TYPE "UDT_ModuleState"
TITLE = UDT_ModuleState
VERSION : 0.1
//User-defined structure of module states.
   STRUCT
      Configured { ExternalAccessible := 'False'; ExternalVisible := 'False'; ExternalWritable := 'False'} : Bool;   // Module configured
      Exist { ExternalAccessible := 'False'; ExternalVisible := 'False'; ExternalWritable := 'False'} : Bool;   // Module exist
      Error { ExternalAccessible := 'False'; ExternalVisible := 'False'; ExternalWritable := 'False'} : Bool;   // Module has error
   END_STRUCT;

END_TYPE

TYPE "UDT_DeviceState"
TITLE = UDT_DeviceState
VERSION : 0.1
//User-defined structure of device states.
   STRUCT
      Configure { ExternalAccessible := 'False'; ExternalVisible := 'False'; ExternalWritable := 'False'} : Bool;   // Device configured in TIA Portal hardware
      Exist { ExternalAccessible := 'False'; ExternalVisible := 'False'; ExternalWritable := 'False'} : Bool;   // Device physically connected
      Error { ExternalAccessible := 'False'; ExternalVisible := 'False'; ExternalWritable := 'False'} : Bool;   // Device has an error
      ProfinetNumber : UInt;   // Profinet slave number
      HW_ID : UInt;   // Device's HW_ID
      PNDeviceName : String;   // Device's project name
   END_STRUCT;

END_TYPE

TYPE "UDT_ProfinetDevice"
TITLE = UDT_ProfinetDevice
VERSION : 0.1
//User-defined structure of profinet device state.
   STRUCT
      DeviceState : "UDT_DeviceState";   // Device state
      Module { S7_SetPoint := 'False'} : Array[0..31] of "UDT_ModuleState";   // Modules
   END_STRUCT;

END_TYPE

TYPE "UDT_GINWCS"
VERSION : 0.1
   STRUCT
      ActionTaken : String;   // Location code value that describes the actual disposition of the package
      Destination1 : String[20];   // Location code value that describes where the package should go (Diverter Number)
      Destination2 : String[20];   // Location code value that describes where the package should go (Diverter Number)
      Destination3 : String[20];   // Location code value that describes where the package should go (Diverter Number)
      Destination4 : String[20];   // Location code value that describes where the package should go (Diverter Number)
      Destination5 : String[20];   // Location code value that describes where the package should go (Diverter Number)
      ReasonCode : String[2];   // Management Code value that describes the result of attempting to route the package to the Destination
      Barcode1 : String;   // Barcode identifier code
      Barcode2 : String;
      Barcode3 : String;
      Barcode4 : String;
   END_STRUCT;

END_TYPE

TYPE "UDT_ProfinetNetwork"
TITLE = UDT_ProfinetNetwork
VERSION : 0.1
//User-defined structure of profinet network state.
   STRUCT
      DeviceStatus : Array[0..512] of "UDT_ProfinetDevice";   // Profinet device status
   END_STRUCT;

END_TYPE

TYPE "UDT_GINWES"
VERSION : 0.1
   STRUCT
      Barcode : String[40];
   END_STRUCT;

END_TYPE

TYPE "UDT_GINDHL"
VERSION : 0.1
   STRUCT
      ObjectID : String[10];   // Object ID
      VID : String[16];   // Virtual Item Identifier (VID)
      PieceID : String[40];   // Piece ID barcodes
      SortStrategy : String[1];   // Sort Strategy 1 - Highest priority available , 2 - Nearest
      ParcelReject { ExternalAccessible := 'False'; ExternalVisible := 'False'; ExternalWritable := 'False'} : Bool;   // True - Parcel reject
      Destination : Array[1..6] of Struct   // Destination
         ID : UInt;   // ID
         SortCommandActive { ExternalAccessible := 'False'; ExternalVisible := 'False'; ExternalWritable := 'False'} : Bool;   // Sort command
         ParcelSorted { ExternalAccessible := 'False'; ExternalVisible := 'False'; ExternalWritable := 'False'} : Bool;   // Parcel sorted
         Rejected { ExternalAccessible := 'False'; ExternalVisible := 'False'; ExternalWritable := 'False'} : Bool;   // Parcel rejected
         Reason : Int;   // Reason
      END_STRUCT;
      ParcelLocation : Struct   // Parcel Location
         Current : UInt;   // Current
         Last : UInt;   // Last
         Sort : UInt;   // Sort
      END_STRUCT;
      MFCMessage : Struct   // MFC Sort messages
         Sent : Struct   // Messages sent from the PLC to the MFC system
            SortResult { ExternalAccessible := 'False'; ExternalVisible := 'False'; ExternalWritable := 'False'} : Bool;   // Message Sort Result
            VIDResponse { ExternalAccessible := 'False'; ExternalVisible := 'False'; ExternalWritable := 'False'} : Bool;   // Message VID Response
            ScanReset { ExternalAccessible := 'False'; ExternalVisible := 'False'; ExternalWritable := 'False'} : Bool;   // Message Scan Reset
            XrayResult { ExternalAccessible := 'False'; ExternalVisible := 'False'; ExternalWritable := 'False'} : Bool;   // Message Xray result
            ParcelRegInfo { ExternalAccessible := 'False'; ExternalVisible := 'False'; ExternalWritable := 'False'} : Bool;   // Message Xray registration info
         END_STRUCT;
         Received : Struct   // Messages received from the MFC system to the PLC
            RejectParcel { ExternalAccessible := 'False'; ExternalVisible := 'False'; ExternalWritable := 'False'} : Bool;   // Message Reject Parcel
            Destination { ExternalAccessible := 'False'; ExternalVisible := 'False'; ExternalWritable := 'False'} : Bool;   // Message Destination
            DestinationResent { ExternalAccessible := 'False'; ExternalVisible := 'False'; ExternalWritable := 'False'} : Bool;   // Message Destination Resent
            TemporaryParcelIdentifier { ExternalAccessible := 'False'; ExternalVisible := 'False'; ExternalWritable := 'False'} : Bool;   // Message Temporary Parcel Identifier
            XrayRegistrationInfo { ExternalAccessible := 'False'; ExternalVisible := 'False'; ExternalWritable := 'False'} : Bool;
         END_STRUCT;
      END_STRUCT;
      Xray : Struct   // Xray data structure
         RoutingCode : String[2];   // Routing code
         Group : String[1];   // The group field is used to identify the group of the operator decisions came from in a
         Level : String[1];   // Level field is used to identify which level the operator decision came from in a
         Result : String[1];   // Results can be indicated with the following:A = Accept, R = Reject, U = Unavailable (Timeout), Z = High Threat
         BagIDMessage : Struct   // Message from PLC to Xray
            MessagePrepared { ExternalAccessible := 'False'; ExternalVisible := 'False'; ExternalWritable := 'False'} : Bool;   // The message is prepared and ready to send
            WrongMessageStructure { ExternalAccessible := 'False'; ExternalVisible := 'False'; ExternalWritable := 'False'} : Bool;   // The message has wrong structure
            Sent { ExternalAccessible := 'False'; ExternalVisible := 'False'; ExternalWritable := 'False'} : Bool;   // The message sent by PLC to Xray
            SentTime : String;   // Time when message sent by PLC to Xray
            NotSent { ExternalAccessible := 'False'; ExternalVisible := 'False'; ExternalWritable := 'False'} : Bool;   // The message was not sent from the PLC
            Received { ExternalAccessible := 'False'; ExternalVisible := 'False'; ExternalWritable := 'False'} : Bool;   // The message received by Xray
            TimeReceived : String;   // Time when message received by Xray
            NotReceived { ExternalAccessible := 'False'; ExternalVisible := 'False'; ExternalWritable := 'False'} : Bool;   // The message did not reach Xray
         END_STRUCT;
         DecisionMessage : Struct   // Message from Xray to PLC
            Received { ExternalAccessible := 'False'; ExternalVisible := 'False'; ExternalWritable := 'False'} : Bool;   // The message received by PLC
            ReceivedTime : String;   // The message received by PLC
            NotReceivedOnTime { ExternalAccessible := 'False'; ExternalVisible := 'False'; ExternalWritable := 'False'} : Bool;   // The message did not reach PLC
         END_STRUCT;
      END_STRUCT;
   END_STRUCT;

END_TYPE

TYPE "UDT_GINUPS"
VERSION : 0.1
   STRUCT
      TRKNUM : String[18];   // Tracking number
      PKGUID : String[32];   // Package ID
      MSGID : String[32];   // Message ID
      Length : Int;   // Camera Length in mm
      Width : Int;   // Camera Width in mm
      Height : Int;   // Camera Height in mm
      Weight : DInt;   // Weight in g
      IDCreated { ExternalAccessible := 'False'; ExternalVisible := 'False'; ExternalWritable := 'False'} : Bool;   // Byte 1, Bit 0 - PLCID created or TrayID Read
      DimDataRcv { ExternalAccessible := 'False'; ExternalVisible := 'False'; ExternalWritable := 'False'} : Bool;   // Byte 1, Bit 1 - Package Dimensional Data Received via Camera Scan Data Message
      PkgWrongInduct { ExternalAccessible := 'False'; ExternalVisible := 'False'; ExternalWritable := 'False'} : Bool;   // Byte 1, Bit 2 - Package Did NOT Induct Properly (Non-Tray Systems)
      IDCalcFromCamID { ExternalAccessible := 'False'; ExternalVisible := 'False'; ExternalWritable := 'False'} : Bool;   // Byte 2, Bit 0 - PLCID/TrayID Calculated From CamID
      UnknownParcelID { ExternalAccessible := 'False'; ExternalVisible := 'False'; ExternalWritable := 'False'} : Bool;   // Byte 2, Bit 4 - Unknown Parcel ID
      UndefinedProblem { ExternalAccessible := 'False'; ExternalVisible := 'False'; ExternalWritable := 'False'} : Bool;   // Byte 2, Bit 5 - Un-Defined Problem
      UnrecognizedCmd { ExternalAccessible := 'False'; ExternalVisible := 'False'; ExternalWritable := 'False'} : Bool;   // Byte 2, Bit 6 - Un-recognized command
      SorterInMainteneceMode { ExternalAccessible := 'False'; ExternalVisible := 'False'; ExternalWritable := 'False'} : Bool;   // Byte 2, Bit 7 - Sorter in Maintenance/Commissioning Mode
      DestUserSusp { ExternalAccessible := 'False'; ExternalVisible := 'False'; ExternalWritable := 'False'} : Bool;   // Byte 3, Bit 3 - Destination User Suspended
      SorterNotSynch { ExternalAccessible := 'False'; ExternalVisible := 'False'; ExternalWritable := 'False'} : Bool;   // Byte 3, Bit 6 - Sorter NOT Synchronized (Tilt Tray Systems)
      PkgDetAtVerCheckPoint { ExternalAccessible := 'False'; ExternalVisible := 'False'; ExternalWritable := 'False'} : Bool;   // Byte 4, Bit 0 - Package Detected at Verification Check Point
      ChuteFullAftrAlterDest { ExternalAccessible := 'False'; ExternalVisible := 'False'; ExternalWritable := 'False'} : Bool;   // Byte 4, Bit 7 - Preferred chute full after passed alternate destination
      ChuteNotAvailAfterAlterDest { ExternalAccessible := 'False'; ExternalVisible := 'False'; ExternalWritable := 'False'} : Bool;   // Byte 5, Bit 0 - Preferred chute not available after passed alternate destination
      PLCRedirected { ExternalAccessible := 'False'; ExternalVisible := 'False'; ExternalWritable := 'False'} : Bool;   // Byte 5, Bit 2 - PLC Redirected
      ThreatParcel { ExternalAccessible := 'False'; ExternalVisible := 'False'; ExternalWritable := 'False'} : Bool;   // Threat parcel
   END_STRUCT;

END_TYPE

TYPE "UDT_GINFedEx"
VERSION : 0.1
   STRUCT
      Timestamp : String[17];   // Local time timestamp
      TimeZoneDesignator : String[5];   // Time zone designator
      PackageEntrancePoint : String[14];   // Entrance point, where LLC starts tracking the parcel.
      PackageEntranceState : String[1];   // Entrance state
      PackageExitPoint : String[14];   // Exit point name, where LLC reports the last known tracking point.
      PackageExitState : String[1];   // Exit point state when LLC reports the last known tracking point.
      PalletType : String[2];   // Pallet code for different type of pallets on the market
      Mask : String[1];   // Flag to indicate that a pallet has been mask.
      CellNumber : String[4];   // Tray/Cell number (for loop sorters) or generated by LLC (on line sorters).
      CellsOccupied : String[1];   // Cells occupied by the piece for loop sorters.
      ImageID : String[6];   // Image ID number created by the ADC system.
      ScanUnitType : String[1];   // Scan unit type
      ADCSystemID : String[15];   // Number assigned by the ADC system
      PackageID : String[15];   // Number assigned by the LLC system
      LLCSystemID : String[15];
      HLCPackageID : String[10];   // Unique number for the specific package during it stays in HLC system.
      HLCResultCode : String[16];   // Result code based on processing of the scan event messages.
      ShipmentID : String[6];   // Consignment id of the parcel.
      WeightStatus : String[1];   // Status to indicate if the parcel/pallet has weight on the system.
      ActualDestination : String[6];   // Location code value that describes the actual disposition of the package.
      Destination1 : String[6];   // Location code value that describes where the package should go (Diverter Number).
      Destination2 : String[6];   // Location code value that describes where the package should go (Diverter Number).
      Destination3 : String[6];   // Location code value that describes where the package should go (Diverter Number).
      Destination4 : String[6];   // Location code value that describes where the package should go (Diverter Number).
      Destination5 : String[6];   // Location code value that describes where the package should go (Diverter Number).
      CutOffTimeDestination1 : String[5];   // Cut Off Time in Local Time.
      CutOffTimeDestination2 : String[5];   // Cut Off Time in Local Time.
      CutOffTimeDestination3 : String[5];   // Cut Off Time in Local Time.
      CutOffTimeDestination4 : String[5];   // Cut Off Time in Local Time.
      CutOffTimeDestination5 : String[5];   // Cut Off Time in Local Time.
      ReasonCode1 : String[8];   // Management Code value that describes the result of attempting to route the package to the Destination
      ReasonCode2 : String[8];   // Management Code value that describes the result of attempting to route the package to the Destination
      ReasonCode3 : String[8];   // Management Code value that describes the result of attempting to route the package to the Destination
      ReasonCode4 : String[8];   // Management Code value that describes the result of attempting to route the package to the Destination
      ReasonCode5 : String[8];   // Management Code value that describes the result of attempting to route the package to the Destination
      HLCDataText : String[20];   // Free text for future use.
      Customs : String[1];   // Need to be checked by customs
      DIMSystemID : String[15];   // Identifier of dimensioning system.
      DIMStatus : String[5];   // Basic diagnostic information from the dimensioning system at the moment of the measurement.
      PackageDimLength : String[6];   // Length dimension of package in resolution of dim system.
      PackageDimWidth : String[6];   // Width dimension of package in resolution of dim system.
      PackageDimHeight : String[6];   // Height dimension of package in resolution of dim system.
      DIMUOM : String[2];   // Unit of measure of the package dimensions.
      DimLFTstatusCode : String[8];   // Dimension LFT status code.
      DimConfidence : String[2];   // The level of assurance for the correct dimensions.
      DimensionSource : String[1];   // For combined camera/laser dim acquisition devices. It indicates type of capturing mode
      AlibiDims : String[25];   // Alibi for Dimensions
      SCLSystemID : String[15];   // Identifier of weight scale.
      SCLStatus : String[5];   // Basic diagnostic information from the weight scale system.
      SCLWT : String[6];   // Scale weight of package in resolution of scale system.
      SCLWTUOM : String[2];   // Unit of measurement for Weight
      SCLLFTStatusCode : String[2];   // Scale LFT status code.
      AlibiWeight : String[25];   // Alibi for Weight
      ReasonCode : String[1];   // This code should be used when the SI message has some defect.
      Stackable : String[1];   // If stackable recognition is enabled, Y or N
      Stickerstype : String[2];   // When optical recognition is used to sort
      FlyingDocument : String[1];   // Status to confirm if the document/flyer is prone to fly off the sorter.
      ModeofOperation : String[1];   // Camera Tunnel operational mode format:
      CameraHeadstatus : String[2];   // Diagnostic information on camera/laser heads performing barcode reads.
      PackageDataTruncated : String[1];   // Y = Full length of barcode data exceeds 9999 bytes, data truncated
      TotalBarcodeDataLength : String[4];   // Length of all barcode data that was sent in bytes;
      Barcode1Identification : String[3];   // Barcode identifier code.
      Barcode1status : String[2];   // Barcode confidence factor
      Barcode1datalength : String[4];   // String length of barcode data in bytes; inclusive of this field. Use 0054 as a fixed value
      Barcode1data : String[50];   // Highest priority barcode
      Barcode2Identification : String[3];   // Barcode identifier code.
      Barcode2status : String[2];   // Barcode confidence factor
      Barcode2datalength : String[4];   // String length of barcode data in bytes; inclusive of this field. Use 0054 as a fixed value
      Barcode2data : String[50];   // Highest priority barcode
      Barcode3Identification : String[3];   // Barcode identifier code.
      Barcode3status : String[2];   // Barcode confidence factor
      Barcode3datalength : String[4];   // String length of barcode data in bytes; inclusive of this field. Use 0054 as a fixed value
      Barcode3data : String[50];   // Highest priority barcode
      BarcodeIdentification : String[3];   // Barcode identifier code.
      Barcodestatus : String[2];   // Barcode confidence factor
      Barcodedatalength : String[4];   // String length of barcode data in bytes
      Barcodedata : String[50];   // Sortation barcode
      CustomerID : DInt;   // 6 digits SequentialID (NNNNNN)
      AreaNumber : String[2];   // Package Sequence ID "Area Number"
      PurgeEnabled { ExternalAccessible := 'False'; ExternalVisible := 'False'; ExternalWritable := 'False'} : Bool;   // Purge enabled for parcel: destination overwritten with Purge destination
   END_STRUCT;

END_TYPE

TYPE "UDT_GINStandard"
VERSION : 0.1
   STRUCT
      Destination : Array[0..20] of DInt;   // Destination
      Identification : Struct   // Barcode identification
         GoodRead { ExternalAccessible := 'False'; ExternalVisible := 'False'; ExternalWritable := 'False'} : Bool;   // Barcode read was succesful
         NoRead { ExternalAccessible := 'False'; ExternalVisible := 'False'; ExternalWritable := 'False'} : Bool;   // Barcode read was unsuccesful
         MultiRead { ExternalAccessible := 'False'; ExternalVisible := 'False'; ExternalWritable := 'False'} : Bool;   // Multiple Barcodes were detected
         Barcode : Array[0..10] of Char;   // Barcode values
      END_STRUCT;
      GinAssigned { ExternalAccessible := 'False'; ExternalVisible := 'False'; ExternalWritable := 'False'} : Bool;   // GIN is assigned to package
      Lost { ExternalAccessible := 'False'; ExternalVisible := 'False'; ExternalWritable := 'False'} : Bool;   // Lost in tracking
      Length : Int;   // Length in mm
      Width : Int;   // Width in mm
      Height : Int;   // Height in mm
      Weight : DInt;   // Weight in g
      PkgTooLong { ExternalAccessible := 'False'; ExternalVisible := 'False'; ExternalWritable := 'False'} : Bool;   // Package is too long
      PkgTooSmall { ExternalAccessible := 'False'; ExternalVisible := 'False'; ExternalWritable := 'False'} : Bool;   // Package is too small
      PkgTooHigh { ExternalAccessible := 'False'; ExternalVisible := 'False'; ExternalWritable := 'False'} : Bool;   // Package is too high
      PkgOverWeight { ExternalAccessible := 'False'; ExternalVisible := 'False'; ExternalWritable := 'False'} : Bool;   // Package is over weight
      TrailingGap : Int;   // Trailing gap size in cm between the package
      LeadingGap : Int;   // Leading gap size in cm between the package
      NrOfRecirculations : Int;   // Number of recirculations
      DestReqSend { ExternalAccessible := 'False'; ExternalVisible := 'False'; ExternalWritable := 'False'} : Bool;   // Destination request sent to high level
      DestRcv { ExternalAccessible := 'False'; ExternalVisible := 'False'; ExternalWritable := 'False'} : Bool;   // Destination received from high level
      SortStatus : Struct   // Sort status of the package
         DivertDestination : Int;   // Destination to which the package is diverted
         GoodDivert { ExternalAccessible := 'False'; ExternalVisible := 'False'; ExternalWritable := 'False'} : Bool;   // Package diverted
         FailedDivert { ExternalAccessible := 'False'; ExternalVisible := 'False'; ExternalWritable := 'False'} : Bool;   // Package failed to divert
         NoDivert : Bool := TRUE;   // Divert is not activated
         NoDivertCause : Struct   // Cause for no divert
            ChuteJam { ExternalAccessible := 'False'; ExternalVisible := 'False'; ExternalWritable := 'False'} : Bool;   // Chute is jammed
            ChuteFull { ExternalAccessible := 'False'; ExternalVisible := 'False'; ExternalWritable := 'False'} : Bool;   // Chute is full
            NoRTR { ExternalAccessible := 'False'; ExternalVisible := 'False'; ExternalWritable := 'False'} : Bool;   // Downstream conveyor is not ready to receive
            DestDisabled { ExternalAccessible := 'False'; ExternalVisible := 'False'; ExternalWritable := 'False'} : Bool;   // Destination is disabled
            TrayDisabled { ExternalAccessible := 'False'; ExternalVisible := 'False'; ExternalWritable := 'False'} : Bool;   // Tray is disabled
            SorterNotAtSpeed { ExternalAccessible := 'False'; ExternalVisible := 'False'; ExternalWritable := 'False'} : Bool;   // Sorter is not at speed
            LeadingGapError { ExternalAccessible := 'False'; ExternalVisible := 'False'; ExternalWritable := 'False'} : Bool;   // Gap size with downstream parcel is not enough
            TrailingGapError { ExternalAccessible := 'False'; ExternalVisible := 'False'; ExternalWritable := 'False'} : Bool;   // Gap size with upstream parcel is not enough
            PkgTooHigh { ExternalAccessible := 'False'; ExternalVisible := 'False'; ExternalWritable := 'False'} : Bool;   // Package is too high to divert
            PkgTooLong { ExternalAccessible := 'False'; ExternalVisible := 'False'; ExternalWritable := 'False'} : Bool;   // Package is too long to divert
            DestNotReachable { ExternalAccessible := 'False'; ExternalVisible := 'False'; ExternalWritable := 'False'} : Bool;   // Sort destionation is not reachable
            InvalidDest { ExternalAccessible := 'False'; ExternalVisible := 'False'; ExternalWritable := 'False'} : Bool;   // Sort destination is invalid
            DestTooLate { ExternalAccessible := 'False'; ExternalVisible := 'False'; ExternalWritable := 'False'} : Bool;   // Destination too late
            NoDestRcv { ExternalAccessible := 'False'; ExternalVisible := 'False'; ExternalWritable := 'False'} : Bool;   // Destination not received from high level
         END_STRUCT;
      END_STRUCT;
   END_STRUCT;

END_TYPE

TYPE "UDT_CommonStatus"
TITLE = UDT_CommonStatus
VERSION : 0.1
//User-defined structure of common statuses.
   STRUCT
      SafetyStop { ExternalAccessible := 'False'; ExternalVisible := 'False'; ExternalWritable := 'False'} : Bool;   // Emergancy stop
      Error { ExternalAccessible := 'False'; ExternalVisible := 'False'; ExternalWritable := 'False'} : Bool;   // An error is active
      Warning { ExternalAccessible := 'False'; ExternalVisible := 'False'; ExternalWritable := 'False'} : Bool;   // A warning is active
      ManualRun { ExternalAccessible := 'False'; ExternalVisible := 'False'; ExternalWritable := 'False'} : Bool;   // Running in manual mode
      Manual { ExternalAccessible := 'False'; ExternalVisible := 'False'; ExternalWritable := 'False'} : Bool;   // In manual mode
      Halted { ExternalAccessible := 'False'; ExternalVisible := 'False'; ExternalWritable := 'False'} : Bool;   // Halted
      Dieback { ExternalAccessible := 'False'; ExternalVisible := 'False'; ExternalWritable := 'False'} : Bool;   // In dieback
      Stopped { ExternalAccessible := 'False'; ExternalVisible := 'False'; ExternalWritable := 'False'} : Bool;   // Stopped
      Running { ExternalAccessible := 'False'; ExternalVisible := 'False'; ExternalWritable := 'False'} : Bool;   // Running
      EnergySave { ExternalAccessible := 'False'; ExternalVisible := 'False'; ExternalWritable := 'False'} : Bool;   // In energy saving mode
      AutoON { ExternalAccessible := 'False'; ExternalVisible := 'False'; ExternalWritable := 'False'} : Bool;   // Automatic started
   END_STRUCT;

END_TYPE

TYPE "UDT_FifoStatus"
TITLE = UDT_FifoStatus
VERSION : 0.1
//
//User-defined structure of FC_Fifo function status.
//Version History:
//Date              | Version   | Author         | Remark
//24/05/2019  | 0.1           | K.Pokorski   | first release MHSE TIA 15.1
//24/05/2019  | 0.2           | K.Pokorski   | first release MHSE TIA 15.1
//
   STRUCT
      InvalidMode { ExternalAccessible := 'False'; ExternalVisible := 'False'; ExternalWritable := 'False'} : Bool;   // Invalid mode selected
      InvalidMaxNrOfEntries { ExternalAccessible := 'False'; ExternalVisible := 'False'; ExternalWritable := 'False'} : Bool;   // Invalid maximum number of entries or buffer is not an array
      InvalidTotalEntriesStored { ExternalAccessible := 'False'; ExternalVisible := 'False'; ExternalWritable := 'False'} : Bool;   // Invalid total number of entries
      InvalidNextEntryToWrite { ExternalAccessible := 'False'; ExternalVisible := 'False'; ExternalWritable := 'False'} : Bool;   // Invalid number of next entry to write
      InvalidNextEntryToRead { ExternalAccessible := 'False'; ExternalVisible := 'False'; ExternalWritable := 'False'} : Bool;   // Invalid number of next entry to read
      InvalidDataType { ExternalAccessible := 'False'; ExternalVisible := 'False'; ExternalWritable := 'False'} : Bool;   // Message and buffer element data type inconsistent
      FifoPreFull { ExternalAccessible := 'False'; ExternalVisible := 'False'; ExternalWritable := 'False'} : Bool;   // 90 % of FIFO data buffer capacity reached
      FifoFull { ExternalAccessible := 'False'; ExternalVisible := 'False'; ExternalWritable := 'False'} : Bool;   // FIFO data buffer full
   END_STRUCT;

END_TYPE

DATA_BLOCK "DB_Memory"
TITLE = DB_Memory
{ S7_Optimized_Access := 'TRUE' }
AUTHOR : MHSE
VERSION : 3.0
NON_RETAIN
   VAR
      ClockByte { ExternalAccessible := 'False'; ExternalVisible := 'False'; ExternalWritable := 'False'} : Byte;   // System clock byte
      Clock_10Hz { ExternalAccessible := 'False'; ExternalVisible := 'False'; ExternalWritable := 'False'} : Bool;   // 10 Hz system clock bit
      Clock_5Hz { ExternalAccessible := 'False'; ExternalVisible := 'False'; ExternalWritable := 'False'} : Bool;   // 5 Hz system clock bit
      "Clock_2.5Hz" { ExternalAccessible := 'False'; ExternalVisible := 'False'; ExternalWritable := 'False'} : Bool;   // 2.5 Hz system clock bit
      Clock_2Hz { ExternalAccessible := 'False'; ExternalVisible := 'False'; ExternalWritable := 'False'} : Bool;   // 2 Hz system clock bit
      "Clock_1.25Hz" { ExternalAccessible := 'False'; ExternalVisible := 'False'; ExternalWritable := 'False'} : Bool;   // 1.25 Hz system clock bit
      Clock_1Hz { ExternalAccessible := 'False'; ExternalVisible := 'False'; ExternalWritable := 'False'} : Bool;   // 1 Hz system clock bit
      "Clock_0.625Hz" { ExternalAccessible := 'False'; ExternalVisible := 'False'; ExternalWritable := 'False'} : Bool;   // 0.625 Hz system clock bit
      "Clock_0.5Hz" { ExternalAccessible := 'False'; ExternalVisible := 'False'; ExternalWritable := 'False'} : Bool;   // 0.5 Hz system clock bit
      SystemByte { ExternalAccessible := 'False'; ExternalVisible := 'False'; ExternalWritable := 'False'} : Byte;   // System byte
      OSClockByte { ExternalAccessible := 'False'; ExternalVisible := 'False'; ExternalWritable := 'False'} : Byte;   // One shot of clock pulse
      "OS_0.1sec" { ExternalAccessible := 'False'; ExternalVisible := 'False'; ExternalWritable := 'False'} : Bool;   // One shot every 0.1 sec
      "OS_0.2sec" { ExternalAccessible := 'False'; ExternalVisible := 'False'; ExternalWritable := 'False'} : Bool;   // One shot every 0.2 sec
      "OS_0.4sec" { ExternalAccessible := 'False'; ExternalVisible := 'False'; ExternalWritable := 'False'} : Bool;   // One shot every 0.4 sec
      "OS_0.5sec" { ExternalAccessible := 'False'; ExternalVisible := 'False'; ExternalWritable := 'False'} : Bool;   // One shot every 0.5 sec
      "OS_0.8sec" { ExternalAccessible := 'False'; ExternalVisible := 'False'; ExternalWritable := 'False'} : Bool;   // One shot every 0.8 sec
      OS_1sec { ExternalAccessible := 'False'; ExternalVisible := 'False'; ExternalWritable := 'False'} : Bool;   // One shot every 1 sec
      "OS_1.6sec" { ExternalAccessible := 'False'; ExternalVisible := 'False'; ExternalWritable := 'False'} : Bool;   // One shot every 1.6 sec
      OS_2sec { ExternalAccessible := 'False'; ExternalVisible := 'False'; ExternalWritable := 'False'} : Bool;   // One shot every 2 sec
      PrevCycleTime { ExternalAccessible := 'False'; ExternalVisible := 'False'; ExternalWritable := 'False'} : LReal;   // Previous PLC cycle Time
      RuntimeMem { ExternalAccessible := 'False'; ExternalVisible := 'False'; ExternalWritable := 'False'} : LReal;   // Runtime memory
      FirstScan { ExternalAccessible := 'False'; ExternalVisible := 'False'; ExternalWritable := 'False'} : Bool;   // First scan bit
      DiagStatusUpdate { ExternalAccessible := 'False'; ExternalVisible := 'False'; ExternalWritable := 'False'} : Bool;   // Diagnostic status update
      AlwaysTrue { ExternalAccessible := 'False'; ExternalVisible := 'False'; ExternalWritable := 'False'} : Bool;   // Always True bit
      AlwaysFalse { ExternalAccessible := 'False'; ExternalVisible := 'False'; ExternalWritable := 'False'} : Bool;   // Always False bit
      CommissioningFalse { ExternalAccessible := 'False'; ExternalVisible := 'False'; ExternalWritable := 'False'} : Bool;   // Commissioning always false
      CommissioningTrue { ExternalAccessible := 'False'; ExternalVisible := 'False'; ExternalWritable := 'False'} : Bool;   // Commissioning always true
      ReconnectCommand { ExternalAccessible := 'False'; ExternalVisible := 'False'; ExternalWritable := 'False'} : Bool;   // Reconnect command
      ScanMainRack { ExternalAccessible := 'False'; ExternalVisible := 'False'; ExternalWritable := 'False'} : Bool;   // Trigger to check main rack confiuration
      ScanProfinet { ExternalAccessible := 'False'; ExternalVisible := 'False'; ExternalWritable := 'False'} : Bool;   // Scan profinet bit
      Simulation { ExternalAccessible := 'False'; ExternalVisible := 'False'; ExternalWritable := 'False'} : Bool;   // Simulation
      PN1OK { ExternalAccessible := 'False'; ExternalVisible := 'False'; ExternalWritable := 'False'} : Bool;   // Profinet ok
      "Local~PROFINET_IO-System" { ExternalAccessible := 'False'; ExternalVisible := 'False'; ExternalWritable := 'False'} : HW_ANY;   // HW Intentifier of PN-IO System
      "Local~PROFINET_IO-System_1" { ExternalAccessible := 'False'; ExternalVisible := 'False'; ExternalWritable := 'False'} : HW_ANY;   // HW Intentifier of PN-IOSystem 1
      "Local~PROFINET_IO-System_2" { ExternalAccessible := 'False'; ExternalVisible := 'False'; ExternalWritable := 'False'} : HW_ANY;   // HW Intentifier of PN-IOSystem 2
      "Local~PROFINET_IO-System_3" { ExternalAccessible := 'False'; ExternalVisible := 'False'; ExternalWritable := 'False'} : HW_ANY;   // HW Intentifier of PN-IOSystem 3
      "Local~PROFINET_IO-System_4" { ExternalAccessible := 'False'; ExternalVisible := 'False'; ExternalWritable := 'False'} : HW_ANY;   // HW Intentifier of PN-IOSystem 4
      "Local~PROFINET_IO-System_5" { ExternalAccessible := 'False'; ExternalVisible := 'False'; ExternalWritable := 'False'} : HW_ANY;   // HW Intentifier of PN-IOSystem 5
      "Local~PROFINET_IO-System_6" { ExternalAccessible := 'False'; ExternalVisible := 'False'; ExternalWritable := 'False'} : HW_ANY;   // HW Intentifier of PN-IOSystem 6
      "Local~PROFINET_IO-System_7" { ExternalAccessible := 'False'; ExternalVisible := 'False'; ExternalWritable := 'False'} : HW_ANY;   // HW Intentifier of PN-IOSystem 7
      "Local~PROFINET_IO-System_8" { ExternalAccessible := 'False'; ExternalVisible := 'False'; ExternalWritable := 'False'} : HW_ANY;   // HW Intentifier of PN-IOSystem 8
      "Local~PROFINET_IO-System_9" { ExternalAccessible := 'False'; ExternalVisible := 'False'; ExternalWritable := 'False'} : HW_ANY;   // HW Intentifier of PN-IOSystem 9
   END_VAR


BEGIN

END_DATA_BLOCK

TYPE "UDT_GIN"
VERSION : 0.1
   STRUCT
      General { S7_SetPoint := 'False'} : "UDT_GINStandard";
      FedEx { S7_SetPoint := 'False'} : "UDT_GINFedEx";
      UPS { S7_SetPoint := 'False'} : "UDT_GINUPS";
      DHL { S7_SetPoint := 'False'} : "UDT_GINDHL";
      WCS { S7_SetPoint := 'False'} : "UDT_GINWCS";
      WES { S7_SetPoint := 'False'} : "UDT_GINWES";
   END_STRUCT;

END_TYPE

DATA_BLOCK "DB_ProfinetDiagnostic"
TITLE = DB_ProfinetDiagnostic
{ S7_Optimized_Access := 'TRUE' }
AUTHOR : MHSE
FAMILY : GeneralSystemFunctions
VERSION : 3.0
NON_RETAIN
//Data block to store profinet network diagnostic data.
   VAR
      ProfinetNetworks { ExternalAccessible := 'False'; ExternalVisible := 'False'; ExternalWritable := 'False'; S7_SetPoint := 'False'} : Array[1..10] of "UDT_ProfinetNetwork";
   END_VAR


BEGIN

END_DATA_BLOCK

TYPE "UDT_EventStatistic"
TITLE = UDT_EventStatistic
VERSION : 0.1
//User-defined structure of event statistic data.
   STRUCT
      NumberOfTimes : DInt;   // Number of times the event occurred since last reset
      LastEventSeconds : DInt;   // Number of seconds of the current or last event
      TotalEventSeconds : DInt;   // Total number of seconds the event occurred since last reset
   END_STRUCT;

END_TYPE

TYPE "UDT_FifoHeader"
TITLE = UDT_FifoHeader
VERSION : 0.1
//User-defined structure of FIFO register header information.
   STRUCT
      Status : Struct   // Status bits
         Empty { ExternalAccessible := 'False'; ExternalVisible := 'False'; ExternalWritable := 'False'} : Bool;   // FIFO Empty
         Prefull { ExternalAccessible := 'False'; ExternalVisible := 'False'; ExternalWritable := 'False'} : Bool;   // FIFO Prefull
         Full { ExternalAccessible := 'False'; ExternalVisible := 'False'; ExternalWritable := 'False'} : Bool;   // FIFO Full
      END_STRUCT;
      NextEntryToRead : Int;   // Next FIFO entry to read
      NextEntryToWrite : Int;   // Next FIFO entry to write
      MaxNrOfEntries : Int;   // Maximum number of FIFO entries
      TotalEntriesStored : Int;   // Total number of FIFO entries
   END_STRUCT;

END_TYPE

FUNCTION "FC_GetNrOfArrayEl" : Int
TITLE = FC_GetNrOfArrayEl
{ S7_Optimized_Access := 'TRUE' }
AUTHOR : MHSE
FAMILY : GeneralSystemFunctions
VERSION : 3.0
// ATTRIBUTES
// AUTO_NUMBER = True
// BLOCK_NUMBER = 19
// END_ATTRIBUTES
//Function to get the number of array elements.
   VAR_INPUT
      iv_Array : Variant;   // Input array
   END_VAR

   VAR_TEMP
      ti_NrOfArrayEl : Int;   // Number of array elements
   END_VAR


BEGIN
	(*
	----------------------------------------------------------------------------------------

	Version history:
	Date        | Version   | Author        | Remark
	----------------------------------------------------------------------------------------
	24/05/2019  | 0.1       | L.Klar        | first release MHS TIA 15.1
	24/07/2019  | 2.0       | L.Klar        | 2.0 MHS library release TIA 15.1
	27/08/2019  | 2.1       | K.Pokorski    | Comments adjusted
	12/11/2019  | 3.0       | P.Majka       | 3.0 MHS library release TIA 15.1
	21/02/2023  | 4.0       | F.Baten       | 4.0 Release TIA 17.5
	*)

	REGION 1 – Number of an array elements

	    IF IS_ARRAY(#iv_Array)                                                  // Input variable is an array
	    THEN

	        #ti_NrOfArrayEl := UDINT_TO_INT(CountOfElements(#iv_Array));

	        // Reset array length if the input variable isn't an array
	    ELSE

	        #ti_NrOfArrayEl := 0;

	    END_IF;

	END_REGION

	REGION 2 – Return output

	    #FC_GetNrOfArrayEl := #ti_NrOfArrayEl;

	END_REGION

END_FUNCTION

TYPE "UDT_PNDevice"
VERSION : 0.1
   STRUCT
      PNNetworknumber : Int := 1;   // Number of the profinet network where device exist
      PNDeviceNumber : Int := 0;   // Profinet number of the device
      PNDeviceFound { ExternalAccessible := 'False'; ExternalVisible := 'False'; ExternalWritable := 'False'} : Bool;   // Device found in Profinet structure
   END_STRUCT;

END_TYPE

TYPE "UDT_VfdStatistics"
TITLE = UDT_VFDStatistics_SEW
VERSION : 0.1
//User-defined structure of FB_VFD_SEW_MOVI-C function block statistics.
   STRUCT
      PNSlaveNotOnline : "UDT_EventStatistic";   // Statistics of Profinet slave not online
      PNSlaveError : "UDT_EventStatistic";   // Statistics of a Profinet slave error
      VFDInternalError : "UDT_EventStatistic";   // Statistics of an internal VFD error
      CommunicationErrorMovikit : "UDT_EventStatistic";   // Statistics of a communication error
      Running : "UDT_EventStatistic";   // Statistics for running time
   END_STRUCT;

END_TYPE

TYPE "UDT_Sorter_DownStream_Basic"
VERSION : 0.1
   STRUCT
      ChuteFull { ExternalAccessible := 'False'; ExternalVisible := 'False'; ExternalWritable := 'False'} : Bool;
      ChuteHalfFull { ExternalAccessible := 'False'; ExternalVisible := 'False'; ExternalWritable := 'False'} : Bool;
      ChuteSensorIncongruence { ExternalAccessible := 'False'; ExternalVisible := 'False'; ExternalWritable := 'False'} : Bool;
      ChuteDisabled { ExternalAccessible := 'False'; ExternalVisible := 'False'; ExternalWritable := 'False'} : Bool;
      ChuteJam { ExternalAccessible := 'False'; ExternalVisible := 'False'; ExternalWritable := 'False'} : Bool;
      ChuteFullSensor { ExternalAccessible := 'False'; ExternalVisible := 'False'; ExternalWritable := 'False'} : Bool;
      ChuteHalfFullSensor { ExternalAccessible := 'False'; ExternalVisible := 'False'; ExternalWritable := 'False'} : Bool;
      ChuteJamSensor { ExternalAccessible := 'False'; ExternalVisible := 'False'; ExternalWritable := 'False'} : Bool;
   END_STRUCT;

END_TYPE

TYPE "UDT_ConveyorInterface"
TITLE = UDT_ConveyorInterface
VERSION : 0.1
//User-defined structure of conveyor interface variables.
   STRUCT
      Displacement : Int;   // Displacement per PLC scan [cm] either from position (if available) or speed and time
      SpeedSetpoint : Int;   // Conveyor speed setpoint [mm/s]
      ActualSpeed : Int;   // Conveyors actual speed [mm/s]
      DeltaPosition : Int;   // Read from Conveyor Servo Position [mm] after 1 PLC cycle
      RunFwd { ExternalAccessible := 'False'; ExternalVisible := 'False'; ExternalWritable := 'False'} : Bool;   // Run forward request
      RunRvs { ExternalAccessible := 'False'; ExternalVisible := 'False'; ExternalWritable := 'False'} : Bool;   // Run reverse request
      InternalErrorEncoder { ExternalAccessible := 'False'; ExternalVisible := 'False'; ExternalWritable := 'False'} : Bool;   // Encoder has an error
      InternalErrorVFD { ExternalAccessible := 'False'; ExternalVisible := 'False'; ExternalWritable := 'False'} : Bool;   // VFD has an error
      InternalErrorTracking { ExternalAccessible := 'False'; ExternalVisible := 'False'; ExternalWritable := 'False'} : Bool;   // Tracking has an error
      InternalErrorPEC { ExternalAccessible := 'False'; ExternalVisible := 'False'; ExternalWritable := 'False'} : Bool;   // PEC has an error
      InternalWarningVFD { ExternalAccessible := 'False'; ExternalVisible := 'False'; ExternalWritable := 'False'} : Bool;   // VFD has a warning
      InternalWarningTracking { ExternalAccessible := 'False'; ExternalVisible := 'False'; ExternalWritable := 'False'} : Bool;   // Tracking has a warning
      InternalErrorReset { ExternalAccessible := 'False'; ExternalVisible := 'False'; ExternalWritable := 'False'} : Bool;   // Reset internal errors
      ConfigurationError { ExternalAccessible := 'False'; ExternalVisible := 'False'; ExternalWritable := 'False'} : Bool;   // Configuration error is active
      VFDRunning { ExternalAccessible := 'False'; ExternalVisible := 'False'; ExternalWritable := 'False'} : Bool;   // Motor is running
      VFDatSpeed { ExternalAccessible := 'False'; ExternalVisible := 'False'; ExternalWritable := 'False'} : Bool;   // Motor at speed setpoint
      Disconnected { ExternalAccessible := 'False'; ExternalVisible := 'False'; ExternalWritable := 'False'} : Bool;   // VFD disconnected
      ManualModeActive { ExternalAccessible := 'False'; ExternalVisible := 'False'; ExternalWritable := 'False'} : Bool;   // Covneyor is in manual mode
      ResetStatistics { ExternalAccessible := 'False'; ExternalVisible := 'False'; ExternalWritable := 'False'} : Bool;   // Reset statistics
      HardwareOk { ExternalAccessible := 'False'; ExternalVisible := 'False'; ExternalWritable := 'False'} : Bool;   // Hardware for the Equipment is available and healthy
   END_STRUCT;

END_TYPE

TYPE "UDT_SerialComConfiguration"
VERSION : 0.1
   STRUCT
      Port : UInt;   // "HW identifier" from the serial communication module
      ResponseTime : LTime := LT#0NS;   // Time when Xray should send Decision message [ms]
      SendMessageLength : UInt;   // Length of the message frame send in bytes
      ReceiveMessageLength : UInt;   // Length of the message frame receive in bytes
      GINRangeStart { ExternalAccessible := 'False'; ExternalVisible := 'False'; ExternalWritable := 'False'} : Int;   // GIN range start value
      GINRangeEnd { ExternalAccessible := 'False'; ExternalVisible := 'False'; ExternalWritable := 'False'} : Int;   // GIN range end value
   END_STRUCT;

END_TYPE

FUNCTION "FC_GetDevicePN" : Void
TITLE = FC_GetDevicePN
{ S7_Optimized_Access := 'TRUE' }
AUTHOR : MHSE
VERSION : 3.0
// ATTRIBUTES
// AUTO_NUMBER = True
// BLOCK_NUMBER = 18
// END_ATTRIBUTES
   VAR_INPUT
      is_PNDeviceName : String;   // Name of the device
      ix_SimulationModeActive : Bool;   // True = Simulation mode active
   END_VAR

   VAR_IN_OUT
      iqUDT_PND : "UDT_PNDevice";   // Device found in Profinet structure
   END_VAR

   VAR_TEMP
      ti_NrOfConfiguredPNNetworks : Int;   // Number of networks configured in project
      ti_NrOfDevices : Int;   // Nr of devices is networks
      ti_LcPNNetworkNumber : Int;   // Loop counter to find PN network number
      ti_LcPNDeviceNumber : Int;   // Loop counter to find PN device number
   END_VAR


BEGIN
	(*
	----------------------------------------------------------------------------------------

	Version history:
	Date        | Version   | Author        | Remark
	----------------------------------------------------------------------------------------
	16/09/2019  | 2.3       | F.Baten       | Cut out of 'FB_RIO'
	29/09/2019  | 2.4       | K.Pokorski    | Network seach started from 1 instead 0
	30/09/2019  | 2.5       | K.Pokorski    | Chagne prefixes of temporary varaibles from 'si' to 'ti'
	12/11/2019  | 3.0       | P.Majka       | 3.0 MHS library release TIA 15.1
	21/02/2023  | 4.0       | F.Baten       | 4.0 Release TIA 17.5
	*)

	REGION 1 - Get Device Profinet number
	    // if simulation is disabled
	    IF NOT #ix_SimulationModeActive
	    THEN
	        // And the profinet device is not found yet
	        IF (#is_PNDeviceName <> "DB_ProfinetDiagnostic".ProfinetNetworks[#iqUDT_PND.PNNetworknumber].DeviceStatus[#iqUDT_PND.PNDeviceNumber].DeviceState.PNDeviceName)
	            OR #iqUDT_PND.PNDeviceFound = FALSE
	        THEN
	            #iqUDT_PND.PNDeviceFound := FALSE;

	            // check how many profinet networks are configured
	            #ti_NrOfConfiguredPNNetworks := "FC_GetNrOfArrayEl"("DB_ProfinetDiagnostic".ProfinetNetworks);

	            FOR #ti_LcPNNetworkNumber := 1 TO (#ti_NrOfConfiguredPNNetworks) DO

	                #iqUDT_PND.PNNetworknumber := #ti_LcPNNetworkNumber;

	                // and check how many devices are configured per network
	                #ti_NrOfDevices := "FC_GetNrOfArrayEl"("DB_ProfinetDiagnostic".ProfinetNetworks[#iqUDT_PND.PNNetworknumber].DeviceStatus);

	                // check for each of the devices in the networks if the PN device name is similair to the configured device name
	                FOR #ti_LcPNDeviceNumber := 0 TO (#ti_NrOfDevices - 1) DO

	                    #iqUDT_PND.PNDeviceNumber := #ti_LcPNDeviceNumber;

	                    // set device found when a match is found for the device name in the PN network
	                    IF (#is_PNDeviceName = "DB_ProfinetDiagnostic".ProfinetNetworks[#iqUDT_PND.PNNetworknumber].DeviceStatus[#iqUDT_PND.PNDeviceNumber].DeviceState.PNDeviceName
	                        AND #is_PNDeviceName <> '')
	                    THEN

	                        #iqUDT_PND.PNDeviceFound := TRUE;
	                        EXIT;

	                    END_IF;
	                END_FOR;

	                // exit loop when device name is matching
	                IF #iqUDT_PND.PNDeviceFound
	                THEN

	                    EXIT;

	                END_IF;
	            END_FOR;
	        END_IF;
	    END_IF;

	END_REGION
END_FUNCTION

FUNCTION "FC_Statistics" : Void
TITLE = FC_Statistics
{ S7_Optimized_Access := 'TRUE' }
AUTHOR : MHSE
FAMILY : GeneralSystemFunctions
VERSION : 3.0
// ATTRIBUTES
// AUTO_NUMBER = True
// BLOCK_NUMBER = 26
// END_ATTRIBUTES
//Function to calculate statistics.
   VAR_INPUT
      ix_Reset : Bool;   // Reset statistics data
      ix_Activate : Bool;   // Activete statistics counters
      ix_RTrigActivate : Bool;   // Activation rise trigger
   END_VAR

   VAR_IN_OUT
      iqUDT_Statistics : "UDT_EventStatistic";   // Statistic structure
   END_VAR


BEGIN
	(*
	----------------------------------------------------------------------------------------

	Version history:
	Date        | Version   | Author        | Remark
	----------------------------------------------------------------------------------------
	24/05/2019  | 0.1       | C. Leite      | first release MHS TIA 15.1
	17/07/2019  | 0.2       | A.Nowak       | Add comments
	24/07/2019  | 2.0       | L.Klar        | 2.0 MHS library release TIA 15.1
	27/08/2019  | 2.1       | M.Kurpiers    | Comments adjusted
	04/11/2019  | 2.2       | L.Klar        | 1 second pulse changed from memory bit to DB variable
	12/11/2019  | 3.0       | P.Majka       | 3.0 MHS library release TIA 15.1
	21/02/2023  | 4.0       | F.Baten       | 4.0 Release TIA 17.5
	*)

	REGION 1 - Number of events

	    IF (#ix_RTrigActivate)      // Event occured
	    THEN

	        // Increment the number of times the event occurred and clear the time of the current or last event
	        #iqUDT_Statistics.NumberOfTimes += 1;
	        #iqUDT_Statistics.LastEventSeconds := 0;

	    END_IF;

	END_REGION

	REGION 2 - Event time

	    // 1 shot every 1 sec and activate statistic counter
	    IF ("DB_Memory".OS_1sec AND #ix_Activate)
	    THEN

	        // Increment the time of the current or last event and the time of all events that occured
	        #iqUDT_Statistics.LastEventSeconds += 1;
	        #iqUDT_Statistics.TotalEventSeconds += 1;

	    END_IF;

	END_REGION

	REGION 3 - Data reset


	    IF (#ix_Reset)                                            // Reset statistics data
	    THEN

	        IF (NOT #ix_Activate)                                 // Statistic counter isn't activate
	        THEN

	            // Clear statistics data
	            #iqUDT_Statistics.NumberOfTimes := 0;
	            #iqUDT_Statistics.LastEventSeconds := 0;
	            #iqUDT_Statistics.TotalEventSeconds := 0;

	        ELSE

	            // Write 1 to the number of times the event occurred and clear times
	            #iqUDT_Statistics.NumberOfTimes := 1;
	            #iqUDT_Statistics.LastEventSeconds := 0;
	            #iqUDT_Statistics.TotalEventSeconds := 0;

	        END_IF;

	    END_IF;

	END_REGION
END_FUNCTION

TYPE "UDT_ConveyorCommonConfiguration"
VERSION : 0.1
   STRUCT
      Length : DInt;   // Conveyor length [mm]
      LengthCorrection : DInt;   // Length correction [mm]
   END_STRUCT;

END_TYPE

TYPE "UDT_VfdStatus"
TITLE = UDT_VfdStatus
VERSION : 0.1
//User-defined structure of VFD status.
   STRUCT
      ErrorCode : Int;   // Error code
      SubErrorCode : Int;   // Sub error code
      PNSlaveNotonline : Bool := FALSE;   // Profinet slave is not on line
      PNSlaveError : Bool := FALSE;   // Profinet slave has an error
      InternalError : Bool := FALSE;   // A VFD internal error is active, see error code
      InternalWarning : Bool := FALSE;   // A VFD internal warning is active, see error code
      CommunicationErrorMovikit : Bool := FALSE;   // Communication error with MoviKit
      VFDRunningFeedbackError : Bool := FALSE;   // Motor is not running
      PNSlaveWarning { ExternalAccessible := 'False'; ExternalVisible := 'False'; ExternalWritable := 'False'} : Bool;   // Profinet slave has a warning
   END_STRUCT;

END_TYPE

TYPE "UDT_VFD_MultiControl_PI"
VERSION : 0.1
   STRUCT
      ErrorMotor1 : Bool;   // High = motor error, Low = motor OK
      ErrorMotor2 : Bool := FALSE;   // High = motor error, Low = motor OK
      ErrorMotor3 : Bool := FALSE;   // High = motor error, Low = motor OK
      ErrorMotor4 : Bool := FALSE;   // High = motor error, Low = motor OK
      Reserve5 : Bool;   // Not used
      Reserve6 : Bool := FALSE;   // Not used
      Reserve7 : Bool := FALSE;   // Not used
      Reserve8 : Bool := FALSE;   // Not used
      SpeedMotor1 : SInt;   // Speed 0...100 (0 = stop, 100 = max speed ), negative values indicate reversed direction of rotation
      SpeedMotor2 : SInt;   // Speed 0...100 (0 = stop, 100 = max speed ), negative values indicate reversed direction of rotation
      SpeedMotor3 : SInt;   // Speed 0...100 (0 = stop, 100 = max speed ), negative values indicate reversed direction of rotation
      SpeedMotor4 : SInt;   // Speed 0...100 (0 = stop, 100 = max speed ), negative values indicate reversed direction of rotation
      Reserve10 : Bool := FALSE;   // Not used
      CurrentMotor1 : UInt;   // Average current in mA
      CurrentMotor2 : UInt;   // Average current in mA
      CurrentMotor3 : UInt;   // Average current in mA
      CurrentMotor4 : UInt;   // Average current in mA
      MotorVoltage : UInt;   // Voltage “Motor Power” in mV
      LogicVoltage : UInt;   // Voltage “Power Logic + Sensors” in mV
   END_STRUCT;

END_TYPE

TYPE "UDT_EquipmentControl"
TITLE = UDT_EquipmentControl
VERSION : 0.1
//User-defined structure of equipment control commands.
   STRUCT
      Command : Struct   // Control command
         Start { ExternalAccessible := 'False'; ExternalVisible := 'False'; ExternalWritable := 'False'} : Bool;   // Start conveyor
         Stop { ExternalAccessible := 'False'; ExternalVisible := 'False'; ExternalWritable := 'False'} : Bool;   // Stop conveyor
         Reset { ExternalAccessible := 'False'; ExternalVisible := 'False'; ExternalWritable := 'False'} : Bool;   // Faults reset
         ResetData { ExternalAccessible := 'False'; ExternalVisible := 'False'; ExternalWritable := 'False'} : Bool;   // Statistics reset
         ManualMode { ExternalAccessible := 'False'; ExternalVisible := 'False'; ExternalWritable := 'False'} : Bool;   // Manual mode required
         DisableManualMode { ExternalAccessible := 'False'; ExternalVisible := 'False'; ExternalWritable := 'False'} : Bool;   // Disable manual mode
         AutomaticOn { ExternalAccessible := 'False'; ExternalVisible := 'False'; ExternalWritable := 'False'} : Bool;   // System is started in automatic mode
         StopRequest { ExternalAccessible := 'False'; ExternalVisible := 'False'; ExternalWritable := 'False'} : Bool;
      END_STRUCT;
      Report { S7_SetPoint := 'False'} : "UDT_CommonStatus";   // Conveyors state
      Request : Struct   // Request from equipment
         RestartRequired { ExternalAccessible := 'False'; ExternalVisible := 'False'; ExternalWritable := 'False'} : Bool;   // Restart required from system control
         SignalingRequest { ExternalAccessible := 'False'; ExternalVisible := 'False'; ExternalWritable := 'False'} : Bool;   // Beeper required
         InhibitStop { ExternalAccessible := 'False'; ExternalVisible := 'False'; ExternalWritable := 'False'} : Bool;
      END_STRUCT;
   END_STRUCT;

END_TYPE

DATA_BLOCK "DB_HMIStatusConfiguration"
TITLE = DB_HMIStatusConfiguration
{ S7_Optimized_Access := 'TRUE' }
AUTHOR : MHSE
VERSION : 3.0
NON_RETAIN
   VAR
      FireAlarm : Int;   // Fire alarm active
      SafetyStop : Int;   // Safety stop error status
      Error : Int;   // Error status
      Warning : Int;   // Warning status
      ManualRun : Int;   // Manual run status
      Manual : Int;   // Manual status
      Halted : Int;   // Halted status
      Dieback : Int;   // Die back status
      Stopped : Int;   // Stopped status
      Running : Int;   // Running status
      EnergySave : Int;   // Energy save status
      CommunicationError : Int;   // Communication error status
      CBError : Int;   // CB error status
      ProfinetError : Int;   // Profinet error status
      HardwareError : Int;   // Hardware error status
      VFDNotHealthy : Int;   // VFD noth healthy status
      VFDError : Int;   // VFD error status
      PECJam : Int;   // PEC jam status
      ChuteFull : Int;   // Chute full status
      EncoderError : Int;   // Encoder error status
      TrackingError : Int;   // Tracking error status
      DimensionError : Int;   // Dimension error status
      OperationalError : Int;   // Operational error status
      AutoON : Int;   // Automatic is on
      ChuteHalfFull : Int;   // Disable by operator
      DisableByManagement : Int;   // Disable by management
      GateOpen : Int;   // Manual operated gate is open
      GateClosed : Int;   // Manual operated gate is closed
      GateClosedAndNoOperatorPresent : Int;   // Manual operated gate is closed and no operator is present
      PositionChangeOngoing : Int;   // Lifting device or arm diverter changing position
      BufferMode : Int;   // BufferMode Active
      ContinuousMode : Int;   // ContinuousMode Active
      LabbelingMode : Int;   // LabbelingMode Active
   END_VAR


BEGIN
   FireAlarm := 1;
   SafetyStop := 3;
   Error := 5;
   Warning := 7;
   ManualRun := 9;
   Manual := 11;
   Halted := 13;
   Dieback := 15;
   Stopped := 17;
   Running := 19;
   EnergySave := 21;
   CommunicationError := 23;
   CBError := 25;
   ProfinetError := 27;
   HardwareError := 29;
   VFDNotHealthy := 31;
   VFDError := 33;
   PECJam := 35;
   ChuteFull := 37;
   EncoderError := 39;
   TrackingError := 41;
   DimensionError := 43;
   OperationalError := 45;
   AutoON := 47;
   ChuteHalfFull := 49;
   DisableByManagement := 51;
   GateOpen := 53;
   GateClosed := 55;
   GateClosedAndNoOperatorPresent := 57;
   PositionChangeOngoing := 59;
   BufferMode := 61;
   ContinuousMode := 63;
   LabbelingMode := 65;

END_DATA_BLOCK

FUNCTION_BLOCK "FB_TimerOnOffDelay"
TITLE = FB_TimerOnOffDelay
{ S7_Optimized_Access := 'TRUE' }
AUTHOR : MHSE
FAMILY : GeneralSystemFunctions
VERSION : 3.0
// ATTRIBUTES
// AUTO_NUMBER = True
// BLOCK_NUMBER = 32
// END_ATTRIBUTES
//Function block to generate on/off signal delay.
   VAR_INPUT
      iudi_OnDelayTime { ExternalAccessible := 'False'; ExternalVisible := 'False'; ExternalWritable := 'False'} : UDInt;   // On delay time [ms]
      iudi_OffDelayTime { ExternalAccessible := 'False'; ExternalVisible := 'False'; ExternalWritable := 'False'} : UDInt;   // Off delay time [ms]
      ix_SignalToDelay { ExternalAccessible := 'False'; ExternalVisible := 'False'; ExternalWritable := 'False'} : Bool;   // Input signal to be delayed
      ix_Enable { ExternalAccessible := 'False'; ExternalVisible := 'False'; ExternalWritable := 'False'} : Bool := TRUE;   // Timer Enable
   END_VAR

   VAR_OUTPUT
      qlr_ActualTime { ExternalAccessible := 'False'; ExternalVisible := 'False'; ExternalWritable := 'False'} : LReal;   // Actual time
      qx_DelayedSignal { ExternalAccessible := 'False'; ExternalVisible := 'False'; ExternalWritable := 'False'} : Bool;   // Delayed signal output
   END_VAR

   VAR
      s_R_TRIG_Signal {InstructionName := 'R_TRIG'; LibVersion := '1.0'; ExternalAccessible := 'False'; ExternalVisible := 'False'; ExternalWritable := 'False'; S7_SetPoint := 'False'} : R_TRIG;   // Siemens "R_Trig" - to prepare the rising edge trigger on "ix_SignalToDelay" signal
      s_F_TRIG_Signal {InstructionName := 'F_TRIG'; LibVersion := '1.0'; ExternalAccessible := 'False'; ExternalVisible := 'False'; ExternalWritable := 'False'; S7_SetPoint := 'False'} : F_TRIG;   // Siemens "F_Trig" - to prepare the falling edge trigger on "ix_SignalToDelay" signal
   END_VAR
   VAR RETAIN
      slr_ActualDelayTime { ExternalAccessible := 'False'; ExternalVisible := 'False'; ExternalWritable := 'False'} : LReal;   // Actual delay time [ms]
   END_VAR


BEGIN
	(*
	----------------------------------------------------------------------------------------

	Version history:
	Date        | Version   | Author        | Remark
	----------------------------------------------------------------------------------------
	24/05/2019  | 0.1       | L.Klar        | first release MHS TIA 15.1
	24/07/2019  | 2.0       | L.Klar        | 2.0 MHS library release TIA 15.1
	26/08/2019  | 2.1       | M.Kurpiers    | Comments adjusted
	04/11/2019  | 2.2       | L.Klar        | Prevoius cycle scan changed from memory to DB variable
	12/11/2019  | 3.0       | P.Majka       | 3.0 MHS library release TIA 15.1
	21/02/2023  | 4.0       | F.Baten       | 4.0 Release TIA 17.5
	*)

	REGION Step 1 – Input signal edge detection

	    #s_R_TRIG_Signal(CLK := #ix_SignalToDelay);


	    #s_F_TRIG_Signal(CLK := #ix_SignalToDelay);

	END_REGION

	REGION Step 2 – Actual delay time initialization

	    IF (#s_R_TRIG_Signal.Q OR #s_F_TRIG_Signal.Q)           // Input signal changed
	    THEN

	        #slr_ActualDelayTime := 0;

	    END_IF;

	END_REGION

	REGION Step 3 – On/Off delay time calculation


	    IF (#ix_SignalToDelay                                       // Signal to be delayed is active
	        AND #ix_Enable)                                         // Ttimer enabled
	    THEN

	        // Timer on
	        IF (#slr_ActualDelayTime >= #iudi_OnDelayTime)
	        THEN

	            #qx_DelayedSignal := TRUE;

	        ELSE

	            #slr_ActualDelayTime += "DB_Memory".PrevCycleTime;

	        END_IF;

	    END_IF;

	    // Timer off
	    IF (NOT #ix_SignalToDelay                                   // Signal to delay is not active
	        AND #ix_Enable)                                         // Timer is enabled
	    THEN

	        IF (#slr_ActualDelayTime >= #iudi_OffDelayTime)
	        THEN

	            #qx_DelayedSignal := FALSE;

	        ELSE

	            #slr_ActualDelayTime += "DB_Memory".PrevCycleTime;

	        END_IF;

	    END_IF;

	END_REGION

	REGION Step 4 – Actual time

	    #qlr_ActualTime := #slr_ActualDelayTime;

	END_REGION
END_FUNCTION_BLOCK

TYPE "UDT_ConnectStatus"
VERSION : 0.1
   STRUCT
      Status : Int;   // Status number
      Specific : Struct   // Specific status structure
         Connected { ExternalAccessible := 'False'; ExternalVisible := 'False'; ExternalWritable := 'False'} : Bool;   // Connected
         CommunicationFault { ExternalAccessible := 'False'; ExternalVisible := 'False'; ExternalWritable := 'False'} : Bool;   // Communication fault
      END_STRUCT;
   END_STRUCT;

END_TYPE

TYPE "UDT_VFD_MultiControl_Configuration"
TITLE = UDT_VFD_Configuration
VERSION : 0.1
//User-defined structure oparameters.
   STRUCT
      MaximumSpeed : Real;   // Maximum speed [mm/s]
      VFDRampUpTime : UDInt;   // VFD ramp up time for monitoring starting [ms]
      VFDRampDownTime : UDInt;   // VFD ramp up time for monitoring stopping [ms]
      SpeedSetpointWindow : Int := 5;   // VFD speed setpoint window (tolerance) [mm/s]
      VFDPNDeviceName : String;   // VFD's Profinet device name
      CorrectionFactor : Real := 1.0;   // Motor factor to correct diagonal mounting (1.0 = straight, standard)
      DirectionReversal : Bool;   // If true, direction will be swapped
      InterlockFwd : Bool;   // False when turning in forward direction is not possible / allowed
      InterlockRvs : Bool;   // False when turning in reverse direction is not possible / allowed
      MinimumCurrentWhenRunninng : UInt;   // Minimum current from motor when it is running. This setting is used to detect that motor is not running when PLC is sending start command
      AutoReset : Bool;
      TimePNErrorMasking : UDInt := 30000;   // Time how long the PN error will be masked, active if AutoReset is True.
   END_STRUCT;

END_TYPE

FUNCTION "FC_StringToTime" : Void
TITLE = FC_StringToTime
{ S7_Optimized_Access := 'TRUE' }
AUTHOR : MHSE
FAMILY : GeneralSystemFunctions
VERSION : 3.0
// ATTRIBUTES
// AUTO_NUMBER = True
// BLOCK_NUMBER = 27
// END_ATTRIBUTES
//Function to convert date in string format to the DTL.
   VAR_INPUT
      is_StringTime : String;   // Input string with date
   END_VAR

   VAR_OUTPUT
      qt_Date {InstructionName := 'DTL'; LibVersion := '1.0'} : DTL;   // Output Date in DTL
   END_VAR

   VAR_TEMP
      ts_DateInt : Struct   // Temp partial date in integer
         Year : UInt;
         Month : USInt;
         Day : USInt;
         Hour : USInt;
         Minute : USInt;
         Second : USInt;
         Millisecond : UDInt;
      END_STRUCT;
      ts_DateString : Struct   // Temp partial date in string
         Hour : String[2];
         Minute : String[2];
         Second : String[2];
         Millisecond : String[3];
      END_STRUCT;
   END_VAR

   VAR CONSTANT
      ci_StringLength2 : Int := 2;   // Length of the part of the string
      ci_StringLength3 : Int := 3;   // Length of the part of the string
      ci_StringPosition1 : Int := 1;   // Position of the first caracter inside the string
      ci_StringPosition4 : Int := 4;   // Position of the first caracter inside the string
      ci_StringPosition7 : Int := 7;   // Position of the first caracter inside the string
      ci_StringPosition10 : Int := 10;   // Position of the first caracter inside the string
      cw_FormatZero : Word := 0;   // Simple value format
      Ci_Year : UInt := 1970;   // Fixed year 1970, start value dtl
      ci_Month : USInt := 1;   // Fixed month 1, start value dtl
      ci_Day : USInt := 1;   // Fixed day 1, start value dtl
   END_VAR


BEGIN
	(*
	----------------------------------------------------------------------------------------

	Version history:
	Date        | Version   | Author        | Remark
	----------------------------------------------------------------------------------------
	24/05/2019  | 0.1       | K.Pokorski    | first release MHS TIA 15.1
	26/06/2019  | 0.2       | M.Kurpiers    | Change in region 1 P:=3 -> P:=4
	24/07/2019  | 2.0       | L.Klar        | 2.0 MHS library release TIA 15.1
	26/07/2019  | 2.1       | M.Kurpiers    | Comments adjusted
	12/11/2019  | 3.0       | P.Majka       | 3.0 MHS library release TIA 15.1
	16/02/2023  | 3.1       | F.Baten       | Added constants
	21/02/2023  | 4.0       | F.Baten       | 4.0 Release TIA 17.5
	*)

	REGION 1 - Separation different part of the date

	    // Separation different part of the date from the data string and saving it to the structure
	    #ts_DateString.Hour := MID(IN := #is_StringTime,
	                               L := #ci_StringLength2,
	                               P := #ci_StringPosition1);               // Separating an hour from the date string
	    #ts_DateString.Minute := MID(IN := #is_StringTime,
	                                 L := #ci_StringLength2,
	                                 P := #ci_StringPosition4);             // Separating a minute from the date string
	    #ts_DateString.Second := MID(IN := #is_StringTime,
	                                 L := #ci_StringLength2,
	                                 P := #ci_StringPosition7);             // Separating a second from the date string
	    #ts_DateString.Millisecond := MID(IN := #is_StringTime,
	                                      L := #ci_StringLength3,
	                                      P := #ci_StringPosition10);       // Separating a millisecond from the date string

	END_REGION

	REGION 2 - Conversion string to integer

	    STRG_VAL(IN := #ts_DateString.Hour,                         // Conversion a hour from string
	             FORMAT := #cw_FormatZero,                          // Simple value format
	             P := INT_TO_UINT(#ci_StringPosition1),             // First position in string
	             OUT => #ts_DateInt.Hour);                          // Integer temporary variable
	    // Conversion a minute from string
	    STRG_VAL(IN := #ts_DateString.Minute,
	             FORMAT := #cw_FormatZero,
	             P := INT_TO_UINT(#ci_StringPosition1),
	             OUT => #ts_DateInt.Minute);
	    // Conversion a second from string
	    STRG_VAL(IN := #ts_DateString.Second,
	             FORMAT := #cw_FormatZero,
	             P := INT_TO_UINT(#ci_StringPosition1),
	             OUT => #ts_DateInt.Second);
	    // Conversion a milisecond from string
	    STRG_VAL(IN := #ts_DateString.Millisecond,
	             FORMAT := #cw_FormatZero,
	             P := INT_TO_UINT(#ci_StringPosition1),
	             OUT => #ts_DateInt.Millisecond);

	END_REGION

	REGION 3 - Combine integer to "DTL" data type and setting output

	    // Move parts of the date to the DTL output structure
	    #qt_Date.YEAR := #Ci_Year;
	    #qt_Date.MONTH := #ci_Month;
	    #qt_Date.DAY := #ci_Day;
	    #qt_Date.HOUR := #ts_DateInt.Hour;
	    #qt_Date.MINUTE := #ts_DateInt.Minute;
	    #qt_Date.SECOND := #ts_DateInt.Second;
	    #qt_Date.NANOSECOND := #ts_DateInt.Millisecond * 1000000;

	END_REGION
END_FUNCTION

TYPE "UDT_MessageV2"
TITLE = UDT_Message
VERSION : 0.1
//User-defined structure of the message characters array.
   STRUCT
      Bytes : Array[0..499] of Byte;   // Message byte
   END_STRUCT;

END_TYPE

DATA_BLOCK "DB_GIN"
TITLE = DB_GIN
{ S7_Optimized_Access := 'TRUE' }
AUTHOR : MHSE
FAMILY : GeneralSystemFunctions
VERSION : 3.0
NON_RETAIN
//Data block to store parcels informations.
   VAR
      GIN { ExternalAccessible := 'False'; ExternalVisible := 'False'; ExternalWritable := 'False'; S7_SetPoint := 'False'} : Array[1..1] of "UDT_GIN";   // GIN informations - for project remove unneeded customers and extend array bound range to 9999
   END_VAR


BEGIN

END_DATA_BLOCK

TYPE "UDT_MFCSortMessageHeader"
VERSION : 0.1
   STRUCT
      SOM : Byte := 16#FD;   // Start of message
      SourceNode : Byte;   // Source node ID
      DestinationNode : Byte;   // Destination node ID
      SeqNumber : Byte;   // Sequence number
      DataLength : Word;   // Data segment length (bytes)
      NumMsg : Word;   // Number of messages contained in the Data Segment
   END_STRUCT;

END_TYPE

FUNCTION "FC_Fifo" : Void
TITLE = FC_Fifo
{ S7_Optimized_Access := 'TRUE' }
AUTHOR : MHSE
FAMILY : GeneralSystemFunctions
VERSION : 3.0
// ATTRIBUTES
// AUTO_NUMBER = True
// BLOCK_NUMBER = 17
// END_ATTRIBUTES
//Function for controlling FIFO register.
   VAR_INPUT
      ic_Mode : Char;   // Mode selector: "W" - Write; "R" - Read; "C" - Clear (Reset) "S" - Status
   END_VAR

   VAR_OUTPUT
      qUDT_Status : "UDT_FifoStatus";   // FIFO status structure
      qx_Error : Bool;   // Collective error output
      qx_Warning : Bool;   // Collective warning output
   END_VAR

   VAR_IN_OUT
      iqv_Data : Variant;   // Data
      iqUDT_FifoHeader : "UDT_FifoHeader";   // FIFO header
      iqv_DataBuffer : Variant;   // FIFO data buffer
   END_VAR

   VAR_TEMP
      tUDT_Status : "UDT_FifoStatus";   // Status structure
      ti_MoveBLKErrorCode : Int;   // Move_BLK_Variant function return
      tx_HeaderValid : Bool;   // Header valid
   END_VAR


BEGIN
	(*
	----------------------------------------------------------------------------------------

	Version history:
	Date        | Version   | Author        | Remark
	----------------------------------------------------------------------------------------
	24/05/2019  | 0.1       | L.Klar        | first release MHS TIA 15.1
	14/06/2019  | 0.2       | A.Nowak       | Replacement of instruction if for direct write into variable - Region 3 , 4.1 , 4.2 , 4.3 , 4.4 , 8.1  , 8.2
	17/07/2019  | 0.3       | L.Klar        | Status handling changed
	24/07/2019  | 2.0       | L.Klar        | 2.0 MHS library release TIA 15.1
	23/08/2019  | 2.1       | K.Pokorski    | Comments corrected
	27/08/2019  | 2.2       | M.Kurpiers    | Comments adjusted
	27/09/2019  | 2.3       | K.Pokorski    | Variant input included
	01/10/2019  | 2.4       | A.Nowak       | Correct comments and rename regions
	12/11/2019  | 3.0       | P.Majka       | 3.0 MHS library release TIA 15.1
	21/02/2023  | 4.0       | F.Baten       | 4.0 Release TIA 17.5
	*)

	REGION 1 – Diagnostic bits initialization

	    // Clear FIFO statuses
	    #tUDT_Status.FifoFull := FALSE;
	    #tUDT_Status.FifoPreFull := FALSE;

	END_REGION

	REGION 2 – Array's information

	    // If buffer elements type is invalid, set the error
	    #tUDT_Status.InvalidDataType := NOT (TypeOf(#iqv_Data) = TypeOfElements(#iqv_DataBuffer));

	END_REGION

	REGION 3 – Mode validation

	    // Set the mode invalid if selected mode isn't one of the following: W- Write, R - Read, C - Clear, S - Status
	    #tUDT_Status.InvalidMode := #ic_Mode <> 'W'
	    AND #ic_Mode <> 'R'
	    AND #ic_Mode <> 'C'
	    AND #ic_Mode <> 'S';

	END_REGION

	REGION 4 – The header settings checking

	    // The correct mode has been selected and data type is valid
	    IF (NOT #tUDT_Status.InvalidMode
	        AND NOT #tUDT_Status.InvalidDataType)
	    THEN

	        REGION 4.1 – The number of maximum FIFO entries validation

	            // Write the number of array's elements to FIFO header
	            #iqUDT_FifoHeader.MaxNrOfEntries := "FC_GetNrOfArrayEl"(#iqv_DataBuffer);

	            // Set the invalid maximum number of entries error
	            #tUDT_Status.InvalidMaxNrOfEntries := #iqUDT_FifoHeader.MaxNrOfEntries <= 0;

	        END_REGION

	        REGION 4.2 – The number of total FIFO entries validation

	            // Set the invalid total number of entries error
	            #tUDT_Status.InvalidTotalEntriesStored := #iqUDT_FifoHeader.TotalEntriesStored < 0        // The total number of entries is lower than 0
	            OR #iqUDT_FifoHeader.TotalEntriesStored > #iqUDT_FifoHeader.MaxNrOfEntries;               // The total number of entries is greater than the maximum number of entries

	        END_REGION

	        REGION 4.3 – The number of the next entry to write

	            // Set the invalid next entry to write
	            #tUDT_Status.InvalidNextEntryToWrite := #iqUDT_FifoHeader.NextEntryToWrite < 0            // The number of next entry to write is lower than 0
	            OR #iqUDT_FifoHeader.NextEntryToWrite >= #iqUDT_FifoHeader.MaxNrOfEntries;                // The number of next entry to write is greater or equal to the maximum number of entries

	        END_REGION

	        REGION 4.4 – The number of the next entry to read

	            // Set the invalid next entry to read
	            #tUDT_Status.InvalidNextEntryToRead := #iqUDT_FifoHeader.NextEntryToRead < 0              // The number of next entry to read is lower than 0
	            OR #iqUDT_FifoHeader.NextEntryToRead >= #iqUDT_FifoHeader.MaxNrOfEntries;                 // The number of next entry to read is greater or equal to the maximum nr of entries

	        END_REGION

	        REGION 4.5 – FIFO header validation summary

	            // Create collective header error
	            #tx_HeaderValid := NOT #tUDT_Status.InvalidMaxNrOfEntries
	            AND NOT #tUDT_Status.InvalidTotalEntriesStored
	            AND NOT #tUDT_Status.InvalidNextEntryToWrite
	            AND NOT #tUDT_Status.InvalidNextEntryToRead;

	        END_REGION

	    END_IF;

	END_REGION

	REGION 5 – Writing the data into the FIFO buffer

	    IF (#ic_Mode = 'W'                                                                          // Write mode selected
	        AND #tx_HeaderValid                                                                     // FIFO header valid
	        AND NOT #tUDT_Status.InvalidDataType)                                                  // Buffer data type valid
	    THEN


	        IF (#iqUDT_FifoHeader.TotalEntriesStored < #iqUDT_FifoHeader.MaxNrOfEntries)          // Checking total number of stored entries
	        THEN

	            // Move input data to FIFO data buffer
	            #ti_MoveBLKErrorCode := MOVE_BLK_VARIANT(SRC := #iqv_Data,
	                                                     COUNT := 1,
	                                                     SRC_INDEX := 0,
	                                                     DEST_INDEX := #iqUDT_FifoHeader.NextEntryToWrite,
	                                                     DEST => #iqv_DataBuffer);

	            // Increment the number of the next entry to write
	            #iqUDT_FifoHeader.NextEntryToWrite += 1;

	            // Increment the total number of stored entries
	            #iqUDT_FifoHeader.TotalEntriesStored += 1;


	            IF (#iqUDT_FifoHeader.NextEntryToWrite >= #iqUDT_FifoHeader.MaxNrOfEntries)       // Check the number of the next entry to write
	            THEN

	                #iqUDT_FifoHeader.NextEntryToWrite := 0;

	            END_IF;

	        ELSE

	            #tUDT_Status.FifoFull := TRUE;

	        END_IF;

	    END_IF;

	END_REGION

	REGION 6 – Reading the data from the FIFO data buffer

	    IF (#ic_Mode = 'R'                                                                  // Read mode selected
	        AND #tx_HeaderValid                                                             // FIFO header valid
	        AND NOT #tUDT_Status.InvalidDataType)                                           // Buffer data type valid
	    THEN

	        IF (#iqUDT_FifoHeader.TotalEntriesStored > 0)                                   // Checking total number of stored entries
	        THEN

	            // Move the FIFO data to the data output
	            #ti_MoveBLKErrorCode := MOVE_BLK_VARIANT(SRC := #iqv_DataBuffer,
	                                                     COUNT := 1,
	                                                     SRC_INDEX := #iqUDT_FifoHeader.NextEntryToRead,
	                                                     DEST_INDEX := 0,
	                                                     DEST => #iqv_Data);

	            // Increment the number of the next entry to read
	            #iqUDT_FifoHeader.NextEntryToRead += 1;

	            // Decrement the total number of stored entries
	            #iqUDT_FifoHeader.TotalEntriesStored -= 1;

	            IF (#iqUDT_FifoHeader.NextEntryToRead >= #iqUDT_FifoHeader.MaxNrOfEntries)  // Check the number of the next entry to read
	            THEN

	                #iqUDT_FifoHeader.NextEntryToRead := 0;

	            END_IF;

	        END_IF;

	    END_IF;

	END_REGION

	REGION 7 – Clearing the FIFO header

	    IF (#ic_Mode = 'C'                      // Clear mode selected
	        AND #tx_HeaderValid)                // FIFO header valid
	    THEN

	        #iqUDT_FifoHeader.TotalEntriesStored := 0;
	        #iqUDT_FifoHeader.NextEntryToWrite := 0;
	        #iqUDT_FifoHeader.NextEntryToRead := 0;

	    END_IF;

	END_REGION

	REGION 8 – FIFO management status update

	    IF (#tx_HeaderValid)                   // The header is valid
	    THEN

	        REGION 8.1 – FIFO Empty

	            // Set the FIFO empty status bit
	            #iqUDT_FifoHeader.Status.Empty := #iqUDT_FifoHeader.TotalEntriesStored = 0;

	        END_REGION

	        REGION 8.2 – FIFO Full

	            // Set the FIFO full status bit
	            #iqUDT_FifoHeader.Status.Full := #iqUDT_FifoHeader.TotalEntriesStored = #iqUDT_FifoHeader.MaxNrOfEntries;

	        END_REGION

	        REGION 8.3 – FIFO Pre-full

	            IF (#iqUDT_FifoHeader.TotalEntriesStored >= 0.9 * #iqUDT_FifoHeader.MaxNrOfEntries)       // Checking if the number of total stored entries is greater or equal to 90% of the max number of entries
	            THEN

	                // Set the FIFO pre-full status
	                #iqUDT_FifoHeader.Status.Prefull := TRUE;
	                #tUDT_Status.FifoPreFull := TRUE;

	            ELSE

	                #iqUDT_FifoHeader.Status.Prefull := FALSE;

	            END_IF;

	        END_REGION

	    END_IF;

	END_REGION

	REGION 9 – Status

	    REGION 9.1 – Common status update

	        // Collective error output
	        #qx_Error := NOT #tx_HeaderValid
	        OR #tUDT_Status.InvalidMode
	        OR #tUDT_Status.FifoFull
	        OR #tUDT_Status.InvalidDataType;

	        // Collective warning output
	        #qx_Warning := #tUDT_Status.FifoPreFull;

	    END_REGION

	    REGION 9.2 – Status update

	        // Update the outer status structure with internal status structure
	        #qUDT_Status := #tUDT_Status;

	    END_REGION

	END_REGION
END_FUNCTION

FUNCTION_BLOCK "FB_Pulse"
TITLE = FB_Pulse
{ S7_Optimized_Access := 'TRUE' }
AUTHOR : MHSE
FAMILY : GeneralSystemFunctions
VERSION : 3.0
// ATTRIBUTES
// AUTO_NUMBER = True
// BLOCK_NUMBER = 26
// END_ATTRIBUTES
//Function block to generate custom pulse signal.
   VAR_INPUT
      iudi_PulseTime { ExternalAccessible := 'False'; ExternalVisible := 'False'; ExternalWritable := 'False'} : UDInt;   // Pulse time [ms]
   END_VAR

   VAR_OUTPUT
      qx_Pulse { ExternalAccessible := 'False'; ExternalVisible := 'False'; ExternalWritable := 'False'} : Bool;   // Pulse output
   END_VAR

   VAR
      R_TRIG {InstructionName := 'R_TRIG'; LibVersion := '1.0'; ExternalAccessible := 'False'; ExternalVisible := 'False'; ExternalWritable := 'False'; S7_SetPoint := 'False'} : R_TRIG;   // Siemens "R_Trig" - to prepare rising edge trigger on "sx_Pulse" signal
      slr_ActualPulseTime { ExternalAccessible := 'False'; ExternalVisible := 'False'; ExternalWritable := 'False'} : LReal;   // Actual pulse time [ms]
      sx_Pulse { ExternalAccessible := 'False'; ExternalVisible := 'False'; ExternalWritable := 'False'} : Bool;   // Pulse signal
   END_VAR


BEGIN
	(*
	----------------------------------------------------------------------------------------

	Version history:
	Date        | Version   | Author        | Remark
	----------------------------------------------------------------------------------------
	24/05/2019  | 0.1       | K.Pokorski    | first release MHS TIA 15.1
	24/07/2019  | 2.0       | L.Klar        | 2.0 MHS library release TIA 15.1
	27/08/2019  | 2.1       | K.Pokorski    | Comments adjusted
	04/11/2019  | 2.2       | L.Klar        | Prevoius cycle scan changed from memory to DB variable
	12/11/2019  | 3.0       | P.Majka       | 3.0 MHS library release TIA 15.1
	21/02/2023  | 4.0       | F.Baten       | 4.0 Release TIA 17.5
	*)

	REGION 1 - Pulse calculation

	    // Pulse timer on
	    IF (#iudi_PulseTime <= #slr_ActualPulseTime)
	    THEN

	        #sx_Pulse := TRUE;
	        #slr_ActualPulseTime := 0;

	    ELSE

	        #slr_ActualPulseTime += "DB_Memory".PrevCycleTime;
	        #sx_Pulse := FALSE;

	    END_IF;

	END_REGION

	REGION 2 - Pulse output

	    #R_TRIG(CLK := #sx_Pulse,
	            Q => #qx_Pulse);

	END_REGION
END_FUNCTION_BLOCK

TYPE "UDT_ColumnLift_Statistics"
TITLE = UDT_VSUStatistics
VERSION : 0.1
//User-defined structure of FB_VerticalSwitch function block statistics.
   STRUCT
      UpTime : "UDT_EventStatistic";   // VSU up time
      DownTime : "UDT_EventStatistic";   // VSU down time
      ManualMode : "UDT_EventStatistic";
      SwitchingTimeError : "UDT_EventStatistic";
   END_STRUCT;

END_TYPE

TYPE "UDT_SecurityCageStatus"
VERSION : 0.1
   STRUCT
      InfeedMode : Bool;   // Infeed mode
      OutfeedMode : Bool;   // Outfeed mode
   END_STRUCT;

END_TYPE

TYPE "UDT_SHA_StationInterface"
VERSION : 0.1
   STRUCT
      Manned : Bool;
      NumberOfParcel : Int;
      TransferInProgres : Bool;
      Conveyor : Array[1..3] of Struct
         Empty : Bool;
         Occupied : Bool;
         Locked : Bool;
      END_STRUCT;
   END_STRUCT;

END_TYPE

TYPE "UDT_SHAStatus"
VERSION : 0.1
   STRUCT
      Status : Int;   // Status number
      Specific : Struct   // Equipment specific
         HalfFull : Bool;   // Halffull status
         Full : Bool;   // Full status
      END_STRUCT;
   END_STRUCT;

END_TYPE

TYPE "UDT_TrackingMonitor"
VERSION : 0.1
   STRUCT
      Data : Int;
      Position : Int;
      DataLength : Int;
   END_STRUCT;

END_TYPE

TYPE "UDT_TrackingOverview"
VERSION : 0.1
   STRUCT
      TotalObject : Int;
      FillingRate : Int;
   END_STRUCT;

END_TYPE

TYPE "UDT_VFD_MultiControl_Universal_Full"
VERSION : 0.1
   STRUCT
      ErrorMotor1 : Bool;   // High = motor error, Low = motor OK
      ErrorMotor2 : Bool := FALSE;   // High = motor error, Low = motor OK
      ErrorMotor3 : Bool := FALSE;   // High = motor error, Low = motor OK
      ErrorMotor4 : Bool := FALSE;   // High = motor error, Low = motor OK
      Reserve5 : Bool;   // Not used
      Reserve6 : Bool := FALSE;   // Not used
      Reserve7 : Bool := FALSE;   // Not used
      Reserve8 : Bool := FALSE;   // Not used
      SpeedMotor1 : SInt;   // Speed 0...100 (0 = stop, 100 = max speed ), negative values indicate reversed direction of rotation
      SpeedMotor2 : SInt;   // Speed 0...100 (0 = stop, 100 = max speed ), negative values indicate reversed direction of rotation
      SpeedMotor3 : SInt;   // Speed 0...100 (0 = stop, 100 = max speed ), negative values indicate reversed direction of rotation
      SpeedMotor4 : SInt;   // Speed 0...100 (0 = stop, 100 = max speed ), negative values indicate reversed direction of rotation
      Reserve10 : Bool := FALSE;   // Not used
      CurrentMotor1 : UInt;   // Average current in mA
      CurrentMotor2 : UInt;   // Average current in mA
      CurrentMotor3 : UInt;   // Average current in mA
      CurrentMotor4 : UInt;   // Average current in mA
      MotorVoltage : UInt;   // Voltage “Motor Power” in mV
      LogicVoltage : UInt;   // Voltage “Power Logic + Sensors” in mV
   END_STRUCT;

END_TYPE

TYPE "UDT_VFD_MultiControl_IOMode"
VERSION : 0.1
   STRUCT
      ErrorMotor1 : Bool;   // High = motor error, Low = motor OK
      ErrorMotor2 : Bool;   // High = motor error, Low = motor OK
      ErrorMotor3 : Bool;   // High = motor error, Low = motor OK
      ErrorMotor4 : Bool;   // High = motor error, Low = motor OK
      ComFail : Bool;   // True = communication error
      PowerFail : Bool;   // True = supply voltage error
      TempFail : Bool;   // True = temperature too high
      ControlFail : Bool;   // True = control system error
      Error : USInt;   // Actual error state: 1 = ready for operation, 2 = minor error, 3 = severe error.
      LastError : USInt;   // Most recent error
      SpeedMotor1 : SInt;   // Speed 0...100 (0 = stop, 100 = max speed ), negative values indicate reversed direction of rotation
      SpeedMotor2 : SInt;   // Speed 0...100 (0 = stop, 100 = max speed ), negative values indicate reversed direction of rotation
      SpeedMotor3 : SInt;   // Speed 0...100 (0 = stop, 100 = max speed ), negative values indicate reversed direction of rotation
      SpeedMotor4 : SInt;   // Speed 0...100 (0 = stop, 100 = max speed ), negative values indicate reversed direction of rotation
   END_STRUCT;

END_TYPE

TYPE "UDT_SystemControlCommand"
TITLE = UDT_SystemControlCommand
VERSION : 0.1
//User-defined structure of system control commands.
   STRUCT
      Start { ExternalAccessible := 'False'; ExternalVisible := 'False'; ExternalWritable := 'False'} : Bool;   // Start Command from HMI
      Stop { ExternalAccessible := 'False'; ExternalVisible := 'False'; ExternalWritable := 'False'} : Bool;   // Stop command from HMI
      Reset { ExternalAccessible := 'False'; ExternalVisible := 'False'; ExternalWritable := 'False'} : Bool;   // Reset command from HMI
      ResetData { ExternalAccessible := 'False'; ExternalVisible := 'False'; ExternalWritable := 'False'} : Bool;   // Reset data command from HMI
      ResetSafety { ExternalAccessible := 'False'; ExternalVisible := 'False'; ExternalWritable := 'False'} : Bool;   // Reset safety command from HMI
      ManualMode { ExternalAccessible := 'False'; ExternalVisible := 'False'; ExternalWritable := 'False'} : Bool;   // Manual mode command from HMI
   END_STRUCT;

END_TYPE

TYPE "UDT_XbeltExitInterface"
VERSION : 0.1
   STRUCT
      ProductLength : Int;   // Product lenght
      ObjectID : DInt;   // Object ID
      NewObjectID : Bool;   // New Object ID
   END_STRUCT;

END_TYPE

TYPE "UDT_XBeltExitStatus"
VERSION : 0.1
   STRUCT
      ChuteDisabled : Bool;   // Chute disabled
      ChuteJam : Bool;   // Chute jam
      ChuteSensorIncongruence : Bool;   // Chute sensor incongruence
   END_STRUCT;

END_TYPE

TYPE "DownStream_Sorter_Basic"
VERSION : 0.1
   STRUCT
      ReadyToReceive { ExternalAccessible := 'False'; ExternalVisible := 'False'; ExternalWritable := 'False'} : Bool;
      Running { ExternalAccessible := 'False'; ExternalVisible := 'False'; ExternalWritable := 'False'} : Bool;
      Fault { ExternalAccessible := 'False'; ExternalVisible := 'False'; ExternalWritable := 'False'} : Bool;
      Warning { ExternalAccessible := 'False'; ExternalVisible := 'False'; ExternalWritable := 'False'} : Bool;
      HalfFull { ExternalAccessible := 'False'; ExternalVisible := 'False'; ExternalWritable := 'False'} : Bool;
      Full { ExternalAccessible := 'False'; ExternalVisible := 'False'; ExternalWritable := 'False'} : Bool;
   END_STRUCT;

END_TYPE

TYPE "UDT_ABSwitchStatus"
TITLE = UDT_VSUStatus
VERSION : 0.1
//User-defined structure of FB_VerticalSwitch function block status.
   STRUCT
      Status : Int;   // Status number
      Specific : Struct   // Equipment specific warnings and errors
         ReferenceError : Bool;   // Active when more like one position sensor active
         SwitchingTimerError : Bool;   // Switching time error
         LimitSensorUpperPosition : Bool;   // Limit switch for upper position active
         LimitSensorLowerPosition : Bool;   // Limit switch for lower position active
         UpperSwitchAreaError : Bool;   // Upper switching area PEC was activated when moving
         LowerSwitchAreaError : Bool;   // Lower switching area PEC was activated when moving
         UpperPosition : Bool;   // Upper position reached
         LowerPosition : Bool;   // Lower position reached
      END_STRUCT;
   END_STRUCT;

END_TYPE

TYPE "UDT_Outfeed2StatesStatus"
VERSION : 0.1
//User-defined structure of FB_CH03 function block status.
   STRUCT
      Status : Int;   // Status number
      Specific : Struct   // CH02 specific status structure
         ChuteFull : Bool;   // Chute is full status
         ChuteHalfFull : Bool;   // Chute is half full status
         ChuteDisabled : Bool;   // Chute is disabled status
      END_STRUCT;
   END_STRUCT;

END_TYPE

TYPE "Sorter_DownStream_Advanced"
VERSION : 0.1
   STRUCT
      Basic { ExternalAccessible := 'False'; ExternalVisible := 'False'; ExternalWritable := 'False'; S7_SetPoint := 'False'} : "UDT_Sorter_DownStream_Basic";
      DischargedObjectID { ExternalAccessible := 'False'; ExternalVisible := 'False'; ExternalWritable := 'False'} : DInt;
      DischargedPackageLength { ExternalAccessible := 'False'; ExternalVisible := 'False'; ExternalWritable := 'False'} : Int;
      DeletedObjectID { ExternalAccessible := 'False'; ExternalVisible := 'False'; ExternalWritable := 'False'} : DInt;
   END_STRUCT;

END_TYPE

FUNCTION "FC_GetPNPortStatus" : Void
{ S7_Optimized_Access := 'TRUE' }
VERSION : 0.1
// ATTRIBUTES
// AUTO_NUMBER = True
// BLOCK_NUMBER = 20
// END_ATTRIBUTES
   VAR_INPUT
      ii_NumberOfPorts : Int;   //  Number of ports in device
      iUDT_DevicePNInfo : "UDT_PNDevice";   //  PN device info structure
   END_VAR

   VAR_OUTPUT
      qa_PortFault : Array[1..8] of Bool;   //  When TRUE then specific port has a fault
   END_VAR

   VAR_TEMP
      tp_GetDiagInfo {InstructionName := 'DIS'; LibVersion := '1.0'} : DIS;   //  Diagnostic structure
      tp_DeviceGeoAddr {InstructionName := 'GEOADDR'; LibVersion := '1.0'} : GEOADDR;   //  Device pointer structre
      ta_PortFault : Array[1..8] of Bool;   //  When TRUE then port has a fault
      ti_Geo2LogStatus : Int;   //  GEO2LOG status code
      ti_GetDiagStatus : Int;   //  Get_Diag status code
      ti_Log2GeoStatus : Int;   //  LOG2GEO status code
      ti_Loopcounter : Int;   //  Loop counter
      tui_cnt : UInt;   //  Not used
      tdi_PortLaddr : HW_ANY;   //  HW identifier
      ti_PortFault : Bool;   //  At least one port is faulty
      tx_ConfigurationError : Bool;   //  Configuration error occurred
   END_VAR

   VAR CONSTANT
      ci_Area : UInt := 1;   //     Area ID of IO Profinet devices
      ci_HWTYPE : UInt := 5;
      ci_PortSlot : UInt := 0;
      ci_PortSubslot : Word := 16#8000;
   END_VAR


BEGIN
	(*
	----------------------------------------------------------------------------------------

	Version history:
	Date        | Version   | Author        | Remark
	----------------------------------------------------------------------------------------
	03/11/2020  | 3.0       | K.Pokorski    | first release MHS TIA 15.1
	17/12/2020  | 3.1       | K.Pokorski    | Run operation only during error
	21/02/2023  | 4.0       | F.Baten       | 4.0 Release TIA 17.5
	*)

	REGION 1 - Check configuration

	    #tx_ConfigurationError := #ii_NumberOfPorts < 1
	    OR #ii_NumberOfPorts > 8
	    OR NOT #iUDT_DevicePNInfo.PNDeviceFound;

	END_REGION

	REGION 2 - Read profinet network number

	    // Using LOG2GEO profinet network address is read
	    #ti_Log2GeoStatus := LOG2GEO(LADDR := "DB_ProfinetDiagnostic".ProfinetNetworks[#iUDT_DevicePNInfo.PNNetworknumber].DeviceStatus[#iUDT_DevicePNInfo.PNDeviceNumber].DeviceState.HW_ID,
	                                 GEOADDR := #tp_DeviceGeoAddr);

	END_REGION

	REGION 3 - Preparation the device pointer

	    // HWTYPE = 5 - Submodule
	    #tp_DeviceGeoAddr.HWTYPE := #ci_HWTYPE;
	    // AREA = 1 - PROFINET IO
	    #tp_DeviceGeoAddr.AREA := #ci_Area;
	    // SLOT = 0 - Ports are on slot 0
	    #tp_DeviceGeoAddr.SLOT := #ci_PortSlot;
	    // STATION - Profinet number
	    #tp_DeviceGeoAddr.STATION := "DB_ProfinetDiagnostic".ProfinetNetworks[#iUDT_DevicePNInfo.PNNetworknumber].DeviceStatus[#iUDT_DevicePNInfo.PNDeviceNumber].DeviceState.ProfinetNumber;

	END_REGION

	REGION 4 - Checking the port status
	    // If device report error and is available on the PN network
	    IF "DB_ProfinetDiagnostic".ProfinetNetworks[#iUDT_DevicePNInfo.PNNetworknumber].DeviceStatus[#iUDT_DevicePNInfo.PNDeviceNumber].DeviceState.Error
	        AND "DB_ProfinetDiagnostic".ProfinetNetworks[#iUDT_DevicePNInfo.PNNetworknumber].DeviceStatus[#iUDT_DevicePNInfo.PNDeviceNumber].DeviceState.Exist
	        AND NOT #tx_ConfigurationError
	    THEN

	        // Loop through all profinet ports
	        FOR #ti_Loopcounter := 1 TO #ii_NumberOfPorts DO
	            // Reset auxiliary port fault bit
	            #ta_PortFault[#ti_Loopcounter] := FALSE;
	            // SUBSLOT = 16#8000 plus port number (TIA structure to refer to port)
	            #tp_DeviceGeoAddr.SUBSLOT := INT_TO_UINT(WORD_TO_INT(#ci_PortSubslot) + (#ti_Loopcounter));
	            // Using GEO2LOG port address is read
	            #ti_Geo2LogStatus := GEO2LOG(GEOADDR := #tp_DeviceGeoAddr, LADDR => #tdi_PortLaddr);
	            // Using GET_DIAG port status is read
	            #ti_GetDiagStatus := GET_DIAG(MODE := 1, LADDR := #tdi_PortLaddr, CNT_DIAG => #tui_cnt, DIAG := #tp_GetDiagInfo);

	            // Set port fault if all operations do not report any error and port is faulty
	            IF #ti_GetDiagStatus = 0
	                AND #ti_Geo2LogStatus = 0
	                AND #ti_Log2GeoStatus = 0
	                AND #tp_GetDiagInfo.OwnState = 4
	            THEN
	                #ta_PortFault[#ti_Loopcounter] := TRUE;
	            END_IF;
	        END_FOR;
	        // Reset module status if error occurred
	    ELSIF #tx_ConfigurationError
	    THEN
	        FOR #ti_Loopcounter := 1 TO 8 DO
	            #ta_PortFault[#ti_Loopcounter] := FALSE;
	        END_FOR;
	    END_IF;

	END_REGION

	REGION 5 - Write output

	    #qa_PortFault := #ta_PortFault;

	END_REGION


END_FUNCTION

TYPE "UDT_RetractrableRoller_Status"
VERSION : 0.1
   STRUCT
      Status : Int;
      Specific : Struct
         NoHomePosition : Bool;
         RollerError : Bool;
      END_STRUCT;
   END_STRUCT;

END_TYPE

TYPE "UDT_InchingStatus"
VERSION : 0.1
   STRUCT
      Full { ExternalAccessible := 'False'; ExternalVisible := 'False'; ExternalWritable := 'False'} : Bool;   // Conveyor is full
      Active { ExternalAccessible := 'False'; ExternalVisible := 'False'; ExternalWritable := 'False'} : Bool;   // Inching is active
   END_STRUCT;

END_TYPE

TYPE "UDT_Outfeed2StatesStatistics"
VERSION : 0.1
//User-defined structure of FB_CH03 function block statistics.
   STRUCT
      ChuteFull { S7_SetPoint := 'False'} : "UDT_EventStatistic";   // Chute full statistics
      ChuteHalfFull : "UDT_EventStatistic";   // Chute half full statistics
      ChuteDisabled { S7_SetPoint := 'False'} : "UDT_EventStatistic";   // Chute disabled statistics
   END_STRUCT;

END_TYPE

TYPE "UDT_ColumnLiftCommand"
VERSION : 0.1
   STRUCT
      MaintenanceControl : Bool;
   END_STRUCT;

END_TYPE

TYPE "UDT_CodingBeltModesConfiguration"
VERSION : 0.1
   STRUCT
      Infeed : Struct   // Infeed configuration:
         LabellingMode : Bool;   // TRUE when mode can be active
         ContinueMode : Bool;   // TRUE when mode can be active
         BufferMode : Bool;   // TRUE when mode can be active
      END_STRUCT;
      Outfeed : Struct   // Outfeed configuration:
         LabellingMode : Bool;   // TRUE when mode can be active
         ContinueMode : Bool;   // TRUE when mode can be active
         BufferMode : Bool;   // TRUE when mode can be active
      END_STRUCT;
      LabellingMode_ParcelStop : Int;   // Parcel stop position in labeling mode, distance between photocell at the beginning of the belt and parcel end.
   END_STRUCT;

END_TYPE

TYPE "UDT_CodingBeltModesStatus"
VERSION : 0.1
   STRUCT
      Status : Int;
      Specific : Struct
         Infeed_LabellingMode : Bool;
         Infeed_ContinueMode : Bool;
         Infeed_BufferMode : Bool;
         Outfeed_LabellingMode : Bool;
         Outfeed_ContinueMode : Bool;
         Outfeed_BufferMode : Bool;
         GeneralError : Bool;
         ConfigurationError : Bool;
      END_STRUCT;
   END_STRUCT;

END_TYPE

TYPE "UDT_CapacityControlConfiguration"
VERSION : 0.1
   STRUCT
      ChuteLength : DInt;   // Hardcode chute lenght [mm]
      MaxProductLenght : DInt;   // Hardcode maximum product lenght [mm]
      ProductLenghtHalfFull : DInt;   // Hardcode halfull product lenght [mm]
   END_STRUCT;

END_TYPE

TYPE "UDT_BiDirectionalConfiguration"
VERSION : 0.1
   STRUCT
      TimeDelayInfeed : UDInt;   // Delay time to keep the system running before turning it off when request a mode change
      TimeDelayOutfeed : UDInt;   // Delay time to keep the system running before turning it off when request a mode change
   END_STRUCT;

END_TYPE

TYPE "UDT_BiDirectionalStatus"
VERSION : 0.1
   STRUCT
      InfeedModeRequested : Bool;   // Mode change is in progress
      OutfeedModeRequested : Bool;   // Mode change is in progress
      InfeedModeActive : Bool;   // Mode active and system running
      OutfeedModeActive : Bool;   // Mode active and system running
      InfeedModeReady : Bool;   // System is ready to restart, wait for start command
      OutfeedModeReady : Bool;   // System is ready to restart, wait for start command
      ChangingMode : Bool;   // The mode will now be changed
   END_STRUCT;

END_TYPE

TYPE "UDT_BiDirectionalInterface"
VERSION : 0.1
   STRUCT
      RequestToStopOutfeed : Bool;   // Request signal to stop outfeed system
      RequestToStopInfeed : Bool;   // Request signal to stop infeed system
      RequestToStopBidirectional : Bool;   // Request signal to stop bidirectional system
      RequestToSwitchingSystem : Bool;   // Request signal to switching system
      RequestToStopSwitchingSystem : Bool;   // Request signal to stop switching system
      OutfeedStopped : Bool;   // Feedback signal from the Outfeed system
      InfeedStopped : Bool;   // Feedback signal from the Intfeed system
      BidirectionalStopped : Bool;   // Feedback signal from the BiDirectional system
      SwitchingSystemReady : Bool;   // Feedback signal from the Switching system
      ElapsedTime : UDInt;   // Change mode elapsed time [sec]
   END_STRUCT;

END_TYPE

TYPE "UDT_ABSwitchConfiguration"
TITLE = UDT_VSUConfig
VERSION : 0.1
//User-defined structure of VSU parameters.
   STRUCT
      JogNoHornTime : UDInt := 1000;   // Time within jog buttons can be pressed without new startup indication
      SwitchingTime : UDInt;   // Time when switching device sholud reach position [ms]
      NominalSpeedSetPoint : Int;   // Nominal spped for position change [mm/s]
      BrakingSpeedSetpoint : Int;   // Speed after braking PEC [mm/s]
      ManualModeSpeed : Int;   // Speed in manual mode [mm/s]
   END_STRUCT;

END_TYPE

TYPE "UDT_ColumnLift_Status"
TITLE = UDT_VSUStatus
VERSION : 0.1
//User-defined structure of FB_VerticalSwitch function block status.
   STRUCT
      Status : Int;   // Status number
      Specific : Struct   // Equipment specific warnings and errors
         ReferenceError : Bool;   // Active when more like one position sensor active
         SwitchingTimerError : Bool;   // Switching time error
         LimitSensorUpperPosition : Bool;   // Limit switch for upper position active
         LimitSensorLowerPosition : Bool;   // Limit switch for lower position active
         UpperPosition : Bool;   // Upper position reached
         LowerPosition : Bool;   // Lower position reached
         ChuteNotInPosition : Bool;   // The chute is not supported by a column
         MaintenaceModeActive : Bool;
      END_STRUCT;
   END_STRUCT;

END_TYPE

TYPE "UDT_ColumnLift_Configuration"
TITLE = UDT_VSUConfig
VERSION : 0.1
//User-defined structure of VSU parameters.
   STRUCT
      ColumnLiftBase : Bool;   // True when downstair base is normal conveyor ; False when downstair base is Caljan with changing height elevation
      JogNoHornTime : UDInt := 1000;   // Time within jog buttons can be pressed without new startup indication [ms]
      SwitchingTime : UDInt;   // Time when switching device sholud reach position [ms]
      NominalSpeedSetPoint : Int;   // Nominal spped for position change [mm/s]
      ManualModeSpeed : Int;   // Speed in manual mode [mm/s]
   END_STRUCT;

END_TYPE

